LIN {X 0,Y 423.097,Z 216.346,A -85,B 0,C 180,E1 -10151.866,E2 -10151.866} C_VEL
LIN {X 0,Y 422.298,Z 296.98,A -85,B 0,C 180,E1 -10153.256,E2 -10153.256} C_VEL
LIN {X 0,Y 421.712,Z 310.923,A -85,B 0,C 180,E1 -10153.699,E2 -10153.699} C_VEL
LIN {X 0,Y 421.172,Z 322.869,A -85,B 0,C 180,E1 -10154.268,E2 -10154.268} C_VEL
LIN {X 0,Y 420.503,Z 334.151,A -85,B 0,C 180,E1 -10154.987,E2 -10154.987} C_VEL
LIN {X 0,Y 419.836,Z 344.931,A -85,B 0,C 180,E1 -10155.867,E2 -10155.867} C_VEL
LIN {X 0,Y 419.115,Z 356.382,A -85,B 0,C 180,E1 -10157.042,E2 -10157.042} C_VEL
LIN {X 0,Y 418.563,Z 364.963,A -85,B 0,C 180,E1 -10158.131,E2 -10158.131} C_VEL
LIN {X 0,Y 417.991,Z 372.886,A -85,B 0,C 180,E1 -10159.343,E2 -10159.343} C_VEL
LIN {X 0,Y 417.563,Z 380.623,A -85,B 0,C 180,E1 -10160.8,E2 -10160.8} C_VEL
LIN {X 0,Y 417.305,Z 386.839,A -85,B 0,C 180,E1 -10162.258,E2 -10162.258} C_VEL
LIN {X 0,Y 417.13,Z 391.886,A -85,B 0,C 180,E1 -10163.753,E2 -10163.753} C_VEL
LIN {X 0,Y 417.134,Z 395.569,A -85,B 0,C 180,E1 -10165.169,E2 -10165.169} C_VEL
LIN {X 0,Y 417.042,Z 397.521,A -85,B 0,C 180,E1 -10166.136,E2 -10166.136} C_VEL
LIN {X 0,Y 417.114,Z 399.058,A -85,B 0,C 180,E1 -10167.104,E2 -10167.104} C_VEL
LIN {X 0,Y 417.095,Z 400.134,A -85,B 0,C 180,E1 -10168.07,E2 -10168.07} C_VEL
LIN {X 0,Y 417.059,Z 401.099,A -85,B 0,C 180,E1 -10170.001,E2 -10170.001} C_VEL
LIN {X 0,Y 417.06,Z 400.999,A -85,B 0,C 180,E1 -10170.966,E2 -10170.966} C_VEL
LIN {X 0,Y 417.092,Z 400.466,A -85,B 0,C 180,E1 -10171.932,E2 -10171.932} C_VEL
LIN {X 0,Y 417.074,Z 399.531,A -85,B 0,C 180,E1 -10172.899,E2 -10172.899} C_VEL
LIN {X 0,Y 417.101,Z 396.464,A -85,B 0,C 180,E1 -10174.834,E2 -10174.834} C_VEL
LIN {X 0,Y 417.064,Z 393.308,A -85,B 0,C 180,E1 -10176.163,E2 -10176.163} C_VEL
LIN {X 0,Y 417.325,Z 388.427,A -85,B 0,C 180,E1 -10177.743,E2 -10177.743} C_VEL
LIN {X 0,Y 417.698,Z 381.536,A -85,B 0,C 180,E1 -10179.443,E2 -10179.443} C_VEL
LIN {X 0,Y 418.217,Z 374.083,A -85,B 0,C 180,E1 -10180.898,E2 -10180.898} C_VEL
LIN {X 0,Y 418.892,Z 366.504,A -85,B 0,C 180,E1 -10182.107,E2 -10182.107} C_VEL
LIN {X 0,Y 419.495,Z 357.34,A -85,B 0,C 180,E1 -10183.319,E2 -10183.319} C_VEL
LIN {X 0,Y 420.276,Z 347.151,A -85,B 0,C 180,E1 -10184.407,E2 -10184.407} C_VEL
LIN {X 0,Y 421.16,Z 335.937,A -85,B 0,C 180,E1 -10185.362,E2 -10185.362} C_VEL
LIN {X 0,Y 422.016,Z 323.303,A -85,B 0,C 180,E1 -10186.198,E2 -10186.198} C_VEL
LIN {X 0,Y 422.766,Z 310.212,A -85,B 0,C 180,E1 -10186.82,E2 -10186.82} C_VEL
LIN {X 0,Y 423.348,Z 297.267,A -85,B 0,C 180,E1 -10187.232,E2 -10187.232} C_VEL
LIN {X 0,Y 424.197,Z 227.472,A -85,B 0,C 180,E1 -10188.452,E2 -10188.452} C_VEL
LIN {X 0,Y 424.203,Z 214.443,A -85,B 0,C 180,E1 -10188.682,E2 -10188.682} C_VEL
LIN {X 0,Y 420.161,Z 189.661,A -85,B 0,C 180,E1 -10189.327,E2 -10189.327} C_VEL
LIN {X 0,Y 419.865,Z 187.56,A -85,B 0,C 180,E1 -10189.403,E2 -10189.403} C_VEL
LIN {X 0,Y 421.208,Z 166.448,A -85,B 0,C 180,E1 -10193.408,E2 -10193.408} C_VEL
LIN {X 0,Y 421.73,Z 158.765,A -85,B 0,C 180,E1 -10194.885,E2 -10194.885} C_VEL
LIN {X 0,Y 420.332,Z 150.718,A -85,B 0,C 180,E1 -10196.569,E2 -10196.569} C_VEL
LIN {X 0,Y 418.298,Z 141.385,A -85,B 0,C 180,E1 -10198.61,E2 -10198.61} C_VEL
LIN {X 0,Y 418.214,Z 141.395,A -85,B 0,C 180,E1 -10201.396,E2 -10201.396} C_VEL
LIN {X 0,Y 418.268,Z 141.381,A -85,B 0,C 180,E1 -10204.58,E2 -10204.58} C_VEL
LIN {X 0,Y 418.226,Z 141.39,A -85,B 0,C 180,E1 -10207.833,E2 -10207.833} C_VEL
LIN {X 0,Y 418.221,Z 141.387,A -85,B 0,C 180,E1 -10210.949,E2 -10210.949} C_VEL
LIN {X 0,Y 418.211,Z 141.392,A -85,B 0,C 180,E1 -10213.729,E2 -10213.729} C_VEL
LIN {X 0,Y 418.208,Z 141.389,A -85,B 0,C 180,E1 -10216.448,E2 -10216.448} C_VEL
LIN {X 0,Y 418.211,Z 141.393,A -85,B 0,C 180,E1 -10219.133,E2 -10219.133} C_VEL
LIN {X 0,Y 418.24,Z 141.388,A -85,B 0,C 180,E1 -10222.776,E2 -10222.776} C_VEL
LIN {X 0,Y 418.234,Z 141.387,A -85,B 0,C 180,E1 -10226.321,E2 -10226.321} C_VEL
LIN {X 0,Y 418.242,Z 141.384,A -85,B 0,C 180,E1 -10229.728,E2 -10229.728} C_VEL
LIN {X 0,Y 418.222,Z 141.391,A -85,B 0,C 180,E1 -10233.017,E2 -10233.017} C_VEL
LIN {X 0,Y 418.258,Z 141.384,A -85,B 0,C 180,E1 -10236.217,E2 -10236.217} C_VEL
LIN {X 0,Y 418.247,Z 141.38,A -85,B 0,C 180,E1 -10239.337,E2 -10239.337} C_VEL
LIN {X 0,Y 418.256,Z 141.385,A -85,B 0,C 180,E1 -10242.395,E2 -10242.395} C_VEL
LIN {X 0,Y 418.263,Z 141.375,A -85,B 0,C 180,E1 -10245.402,E2 -10245.402} C_VEL
LIN {X 0,Y 418.352,Z 141.368,A -85,B 0,C 180,E1 -10247.386,E2 -10247.386} C_VEL
LIN {X 0,Y 418.366,Z 141.361,A -85,B 0,C 180,E1 -10251.304,E2 -10251.304} C_VEL
LIN {X 0,Y 418.467,Z 141.361,A -85,B 0,C 180,E1 -10254.217,E2 -10254.217} C_VEL
LIN {X 0,Y 418.532,Z 141.347,A -85,B 0,C 180,E1 -10258.076,E2 -10258.076} C_VEL
LIN {X 0,Y 418.405,Z 141.363,A -85,B 0,C 180,E1 -10260.963,E2 -10260.963} C_VEL
LIN {X 0,Y 418.468,Z 141.348,A -85,B 0,C 180,E1 -10262.888,E2 -10262.888} C_VEL
LIN {X 0,Y 418.44,Z 141.359,A -85,B 0,C 180,E1 -10266.478,E2 -10266.478} C_VEL
LIN {X 0,Y 418.377,Z 141.359,A -85,B 0,C 180,E1 -10268.696,E2 -10268.696} C_VEL
LIN {X 0,Y 418.314,Z 141.38,A -85,B 0,C 180,E1 -10271.631,E2 -10271.631} C_VEL
LIN {X 0,Y 418.299,Z 141.37,A -85,B 0,C 180,E1 -10274.597,E2 -10274.597} C_VEL
LIN {X 0,Y 418.28,Z 141.381,A -85,B 0,C 180,E1 -10277.604,E2 -10277.604} C_VEL
LIN {X 0,Y 418.251,Z 141.381,A -85,B 0,C 180,E1 -10280.663,E2 -10280.663} C_VEL
LIN {X 0,Y 418.274,Z 141.376,A -85,B 0,C 180,E1 -10283.782,E2 -10283.782} C_VEL
LIN {X 0,Y 418.268,Z 141.385,A -85,B 0,C 180,E1 -10287.059,E2 -10287.059} C_VEL
LIN {X 0,Y 418.244,Z 141.384,A -85,B 0,C 180,E1 -10290.272,E2 -10290.272} C_VEL
LIN {X 0,Y 418.249,Z 141.382,A -85,B 0,C 180,E1 -10293.677,E2 -10293.677} C_VEL
LIN {X 0,Y 418.241,Z 141.385,A -85,B 0,C 180,E1 -10297.224,E2 -10297.224} C_VEL
LIN {X 0,Y 418.245,Z 141.38,A -85,B 0,C 180,E1 -10299.683,E2 -10299.683} C_VEL
LIN {X 0,Y 418.232,Z 141.38,A -85,B 0,C 180,E1 -10302.321,E2 -10302.321} C_VEL
LIN {X 0,Y 418.239,Z 141.384,A -85,B 0,C 180,E1 -10305.109,E2 -10305.109} C_VEL
LIN {X 0,Y 418.237,Z 141.386,A -85,B 0,C 180,E1 -10307.766,E2 -10307.766} C_VEL
LIN {X 0,Y 418.246,Z 141.386,A -85,B 0,C 180,E1 -10310.621,E2 -10310.621} C_VEL
LIN {X 0,Y 418.247,Z 141.389,A -85,B 0,C 180,E1 -10313.976,E2 -10313.976} C_VEL
LIN {X 0,Y 418.262,Z 141.383,A -85,B 0,C 180,E1 -10317.156,E2 -10317.156} C_VEL
LIN {X 0,Y 418.273,Z 141.384,A -85,B 0,C 180,E1 -10320.895,E2 -10320.895} C_VEL
LIN {X 0,Y 418.345,Z 141.524,A -85,B 0,C 180,E1 -10323.025,E2 -10323.025} C_VEL
LIN {X 0,Y 420.17,Z 150.792,A -85,B 0,C 180,E1 -10325.281,E2 -10325.281} C_VEL
LIN {X 0,Y 420.345,Z 152.604,A -85,B 0,C 180,E1 -10325.696,E2 -10325.696} C_VEL
LIN {X 0,Y 424.762,Z 171.221,A -85,B 0,C 180,E1 -10326.26,E2 -10326.26} C_VEL
LIN {X 0,Y 423.727,Z 259.847,A -85,B 0,C 180,E1 -10327.799,E2 -10327.799} C_VEL
LIN {X 0,Y 423.245,Z 273.544,A -85,B 0,C 180,E1 -10328.237,E2 -10328.237} C_VEL
LIN {X 0,Y 422.763,Z 285.058,A -85,B 0,C 180,E1 -10328.786,E2 -10328.786} C_VEL
LIN {X 0,Y 422.155,Z 296.809,A -85,B 0,C 180,E1 -10329.536,E2 -10329.536} C_VEL
LIN {X 0,Y 421.289,Z 308.537,A -85,B 0,C 180,E1 -10330.509,E2 -10330.509} C_VEL
LIN {X 0,Y 420.515,Z 319.047,A -85,B 0,C 180,E1 -10331.611,E2 -10331.611} C_VEL
LIN {X 0,Y 419.859,Z 328.587,A -85,B 0,C 180,E1 -10332.858,E2 -10332.858} C_VEL
LIN {X 0,Y 419.159,Z 336.843,A -85,B 0,C 180,E1 -10334.188,E2 -10334.188} C_VEL
LIN {X 0,Y 418.482,Z 344.233,A -85,B 0,C 180,E1 -10335.657,E2 -10335.657} C_VEL
LIN {X 0,Y 417.937,Z 350.995,A -85,B 0,C 180,E1 -10337.372,E2 -10337.372} C_VEL
LIN {X 0,Y 417.623,Z 355.433,A -85,B 0,C 180,E1 -10338.84,E2 -10338.84} C_VEL
LIN {X 0,Y 417.337,Z 358.788,A -85,B 0,C 180,E1 -10340.304,E2 -10340.304} C_VEL
LIN {X 0,Y 417.213,Z 361.303,A -85,B 0,C 180,E1 -10341.946,E2 -10341.946} C_VEL
LIN {X 0,Y 416.513,Z 362.24,A -85,B 0,C 180,E1 -10342.743,E2 -10342.743} C_VEL
LIN {X 0,Y 413.581,Z 363.208,A -85,B 0,C 180,E1 -10344.045,E2 -10344.045} C_VEL
LIN {X 0,Y 411.127,Z 363.394,A -85,B 0,C 180,E1 -10345.101,E2 -10345.101} C_VEL
LIN {X 0,Y 410.094,Z 363.129,A -85,B 0,C 180,E1 -10345.917,E2 -10345.917} C_VEL
LIN {X 0,Y 410.022,Z 362.954,A -85,B 0,C 180,E1 -10346.193,E2 -10346.193} C_VEL
LIN {X 0,Y 410.105,Z 362.339,A -85,B 0,C 180,E1 -10347.052,E2 -10347.052} C_VEL
LIN {X 0,Y 410.075,Z 361.229,A -85,B 0,C 180,E1 -10348.035,E2 -10348.035} C_VEL
LIN {X 0,Y 410.201,Z 357.742,A -85,B 0,C 180,E1 -10349.999,E2 -10349.999} C_VEL
LIN {X 0,Y 410.379,Z 353.97,A -85,B 0,C 180,E1 -10351.471,E2 -10351.471} C_VEL
LIN {X 0,Y 410.654,Z 349.089,A -85,B 0,C 180,E1 -10352.942,E2 -10352.942} C_VEL
LIN {X 0,Y 411.139,Z 342.947,A -85,B 0,C 180,E1 -10354.411,E2 -10354.411} C_VEL
LIN {X 0,Y 411.719,Z 335.291,A -85,B 0,C 180,E1 -10355.878,E2 -10355.878} C_VEL
LIN {X 0,Y 412.361,Z 327.463,A -85,B 0,C 180,E1 -10357.097,E2 -10357.097} C_VEL
LIN {X 0,Y 413.07,Z 317.923,A -85,B 0,C 180,E1 -10358.314,E2 -10358.314} C_VEL
LIN {X 0,Y 413.815,Z 307.327,A -85,B 0,C 180,E1 -10359.407,E2 -10359.407} C_VEL
LIN {X 0,Y 414.433,Z 296.178,A -85,B 0,C 180,E1 -10360.323,E2 -10360.323} C_VEL
LIN {X 0,Y 414.947,Z 283.723,A -85,B 0,C 180,E1 -10361.107,E2 -10361.107} C_VEL
LIN {X 0,Y 415.398,Z 271.188,A -85,B 0,C 180,E1 -10361.682,E2 -10361.682} C_VEL
LIN {X 0,Y 415.689,Z 257.936,A -85,B 0,C 180,E1 -10362.076,E2 -10362.076} C_VEL
LIN {X 0,Y 416.741,Z 172.858,A -85,B 0,C 180,E1 -10363.547,E2 -10363.547} C_VEL
LIN {X 0,Y 412.858,Z 152.57,A -85,B 0,C 180,E1 -10364.097,E2 -10364.097} C_VEL
LIN {X 0,Y 412.536,Z 148.394,A -85,B 0,C 180,E1 -10365.057,E2 -10365.057} C_VEL
LIN {X 0,Y 411.291,Z 142.256,A -85,B 0,C 180,E1 -10366.551,E2 -10366.551} C_VEL
LIN {X 0,Y 411.231,Z 142.263,A -85,B 0,C 180,E1 -10369.985,E2 -10369.985} C_VEL
LIN {X 0,Y 411.195,Z 142.262,A -85,B 0,C 180,E1 -10373.147,E2 -10373.147} C_VEL
LIN {X 0,Y 411.236,Z 142.261,A -85,B 0,C 180,E1 -10376.38,E2 -10376.38} C_VEL
LIN {X 0,Y 411.198,Z 142.263,A -85,B 0,C 180,E1 -10379.711,E2 -10379.711} C_VEL
LIN {X 0,Y 411.204,Z 142.261,A -85,B 0,C 180,E1 -10383.154,E2 -10383.154} C_VEL
LIN {X 0,Y 411.189,Z 142.265,A -85,B 0,C 180,E1 -10386.551,E2 -10386.551} C_VEL
LIN {X 0,Y 411.213,Z 142.264,A -85,B 0,C 180,E1 -10389.727,E2 -10389.727} C_VEL
LIN {X 0,Y 411.168,Z 142.266,A -85,B 0,C 180,E1 -10393.132,E2 -10393.132} C_VEL
LIN {X 0,Y 411.161,Z 142.271,A -85,B 0,C 180,E1 -10395.88,E2 -10395.88} C_VEL
LIN {X 0,Y 411.156,Z 142.267,A -85,B 0,C 180,E1 -10398.771,E2 -10398.771} C_VEL
LIN {X 0,Y 411.184,Z 142.266,A -85,B 0,C 180,E1 -10402.025,E2 -10402.025} C_VEL
LIN {X 0,Y 411.196,Z 142.266,A -85,B 0,C 180,E1 -10405.665,E2 -10405.665} C_VEL
LIN {X 0,Y 411.18,Z 142.267,A -85,B 0,C 180,E1 -10409.151,E2 -10409.151} C_VEL
LIN {X 0,Y 411.249,Z 142.256,A -85,B 0,C 180,E1 -10412.521,E2 -10412.521} C_VEL
LIN {X 0,Y 411.201,Z 142.265,A -85,B 0,C 180,E1 -10415.783,E2 -10415.783} C_VEL
LIN {X 0,Y 411.185,Z 142.266,A -85,B 0,C 180,E1 -10418.965,E2 -10418.965} C_VEL
LIN {X 0,Y 411.232,Z 142.259,A -85,B 0,C 180,E1 -10422.084,E2 -10422.084} C_VEL
LIN {X 0,Y 411.24,Z 142.261,A -85,B 0,C 180,E1 -10425.146,E2 -10425.146} C_VEL
LIN {X 0,Y 411.27,Z 142.254,A -85,B 0,C 180,E1 -10428.167,E2 -10428.167} C_VEL
LIN {X 0,Y 411.306,Z 142.252,A -85,B 0,C 180,E1 -10431.154,E2 -10431.154} C_VEL
LIN {X 0,Y 411.405,Z 142.237,A -85,B 0,C 180,E1 -10434.117,E2 -10434.117} C_VEL
LIN {X 0,Y 411.489,Z 142.226,A -85,B 0,C 180,E1 -10438.042,E2 -10438.042} C_VEL
LIN {X 0,Y 411.364,Z 142.245,A -85,B 0,C 180,E1 -10440.979,E2 -10440.979} C_VEL
LIN {X 0,Y 411.416,Z 142.238,A -85,B 0,C 180,E1 -10442.937,E2 -10442.937} C_VEL
LIN {X 0,Y 411.418,Z 142.235,A -85,B 0,C 180,E1 -10445.883,E2 -10445.883} C_VEL
LIN {X 0,Y 411.306,Z 142.252,A -85,B 0,C 180,E1 -10448.846,E2 -10448.846} C_VEL
LIN {X 0,Y 411.27,Z 142.254,A -85,B 0,C 180,E1 -10451.833,E2 -10451.833} C_VEL
LIN {X 0,Y 411.245,Z 142.26,A -85,B 0,C 180,E1 -10454.853,E2 -10454.853} C_VEL
LIN {X 0,Y 411.233,Z 142.258,A -85,B 0,C 180,E1 -10457.916,E2 -10457.916} C_VEL
LIN {X 0,Y 411.185,Z 142.267,A -85,B 0,C 180,E1 -10461.035,E2 -10461.035} C_VEL
LIN {X 0,Y 411.2,Z 142.264,A -85,B 0,C 180,E1 -10464.217,E2 -10464.217} C_VEL
LIN {X 0,Y 411.248,Z 142.256,A -85,B 0,C 180,E1 -10467.478,E2 -10467.478} C_VEL
LIN {X 0,Y 411.18,Z 142.267,A -85,B 0,C 180,E1 -10470.848,E2 -10470.848} C_VEL
LIN {X 0,Y 411.195,Z 142.266,A -85,B 0,C 180,E1 -10474.335,E2 -10474.335} C_VEL
LIN {X 0,Y 411.183,Z 142.266,A -85,B 0,C 180,E1 -10477.975,E2 -10477.975} C_VEL
LIN {X 0,Y 411.155,Z 142.267,A -85,B 0,C 180,E1 -10481.229,E2 -10481.229} C_VEL
LIN {X 0,Y 411.168,Z 142.269,A -85,B 0,C 180,E1 -10484.492,E2 -10484.492} C_VEL
LIN {X 0,Y 411.171,Z 142.271,A -85,B 0,C 180,E1 -10488.196,E2 -10488.196} C_VEL
LIN {X 0,Y 411.217,Z 142.26,A -85,B 0,C 180,E1 -10490.778,E2 -10490.778} C_VEL
LIN {X 0,Y 411.193,Z 142.264,A -85,B 0,C 180,E1 -10494.472,E2 -10494.472} C_VEL
LIN {X 0,Y 411.203,Z 142.26,A -85,B 0,C 180,E1 -10496.875,E2 -10496.875} C_VEL
LIN {X 0,Y 411.23,Z 142.263,A -85,B 0,C 180,E1 -10500.645,E2 -10500.645} C_VEL
LIN {X 0,Y 411.295,Z 142.381,A -85,B 0,C 180,E1 -10502.05,E2 -10502.05} C_VEL
LIN {X 0,Y 413.922,Z 155.94,A -85,B 0,C 180,E1 -10504.884,E2 -10504.884} C_VEL
LIN {X 0,Y 414.049,Z 160.059,A -85,B 0,C 180,E1 -10505.695,E2 -10505.695} C_VEL
LIN {X 0,Y 412.864,Z 177.718,A -85,B 0,C 180,E1 -10509.056,E2 -10509.056} C_VEL
LIN {X 0,Y 412.362,Z 187.731,A -85,B 0,C 180,E1 -10510.925,E2 -10510.925} C_VEL
LIN {X 0,Y 416.291,Z 216.452,A -85,B 0,C 180,E1 -10511.597,E2 -10511.597} C_VEL
LIN {X 0,Y 415.449,Z 296.703,A -85,B 0,C 180,E1 -10513.003,E2 -10513.003} C_VEL
LIN {X 0,Y 414.83,Z 310.629,A -85,B 0,C 180,E1 -10513.452,E2 -10513.452} C_VEL
LIN {X 0,Y 414.247,Z 323.112,A -85,B 0,C 180,E1 -10514.061,E2 -10514.061} C_VEL
LIN {X 0,Y 413.503,Z 335.041,A -85,B 0,C 180,E1 -10514.853,E2 -10514.853} C_VEL
LIN {X 0,Y 412.729,Z 346.51,A -85,B 0,C 180,E1 -10515.832,E2 -10515.832} C_VEL
LIN {X 0,Y 412.066,Z 357.099,A -85,B 0,C 180,E1 -10516.97,E2 -10516.97} C_VEL
LIN {X 0,Y 411.452,Z 366.135,A -85,B 0,C 180,E1 -10518.173,E2 -10518.173} C_VEL
LIN {X 0,Y 410.775,Z 375.155,A -85,B 0,C 180,E1 -10519.652,E2 -10519.652} C_VEL
LIN {X 0,Y 410.4,Z 382.423,A -85,B 0,C 180,E1 -10521.135,E2 -10521.135} C_VEL
LIN {X 0,Y 410.171,Z 388.22,A -85,B 0,C 180,E1 -10522.618,E2 -10522.618} C_VEL
LIN {X 0,Y 410.002,Z 392.777,A -85,B 0,C 180,E1 -10524.098,E2 -10524.098} C_VEL
LIN {X 0,Y 410.041,Z 395.183,A -85,B 0,C 180,E1 -10525.085,E2 -10525.085} C_VEL
LIN {X 0,Y 409.959,Z 397.146,A -85,B 0,C 180,E1 -10526.069,E2 -10526.069} C_VEL
LIN {X 0,Y 410.011,Z 398.696,A -85,B 0,C 180,E1 -10527.053,E2 -10527.053} C_VEL
LIN {X 0,Y 410.023,Z 399.789,A -85,B 0,C 180,E1 -10528.036,E2 -10528.036} C_VEL
LIN {X 0,Y 409.978,Z 400.772,A -85,B 0,C 180,E1 -10530.001,E2 -10530.001} C_VEL
LIN {X 0,Y 409.982,Z 400.682,A -85,B 0,C 180,E1 -10530.983,E2 -10530.983} C_VEL
LIN {X 0,Y 410.019,Z 400.166,A -85,B 0,C 180,E1 -10531.965,E2 -10531.965} C_VEL
LIN {X 0,Y 409.971,Z 399.239,A -85,B 0,C 180,E1 -10532.949,E2 -10532.949} C_VEL
LIN {X 0,Y 410.008,Z 396.194,A -85,B 0,C 180,E1 -10534.917,E2 -10534.917} C_VEL
LIN {X 0,Y 409.999,Z 392.73,A -85,B 0,C 180,E1 -10536.397,E2 -10536.397} C_VEL
LIN {X 0,Y 410.266,Z 388.196,A -85,B 0,C 180,E1 -10537.878,E2 -10537.878} C_VEL
LIN {X 0,Y 410.654,Z 381.341,A -85,B 0,C 180,E1 -10539.606,E2 -10539.606} C_VEL
LIN {X 0,Y 411.219,Z 373.917,A -85,B 0,C 180,E1 -10541.086,E2 -10541.086} C_VEL
LIN {X 0,Y 412.045,Z 364.711,A -85,B 0,C 180,E1 -10542.561,E2 -10542.561} C_VEL
LIN {X 0,Y 412.7,Z 355.159,A -85,B 0,C 180,E1 -10543.793,E2 -10543.793} C_VEL
LIN {X 0,Y 413.608,Z 344.588,A -85,B 0,C 180,E1 -10544.893,E2 -10544.893} C_VEL
LIN {X 0,Y 414.57,Z 332.794,A -85,B 0,C 180,E1 -10545.865,E2 -10545.865} C_VEL
LIN {X 0,Y 415.393,Z 320.17,A -85,B 0,C 180,E1 -10546.653,E2 -10546.653} C_VEL
LIN {X 0,Y 416.117,Z 307.584,A -85,B 0,C 180,E1 -10547.224,E2 -10547.224} C_VEL
LIN {X 0,Y 416.707,Z 294.35,A -85,B 0,C 180,E1 -10547.61,E2 -10547.61} C_VEL
LIN {X 0,Y 417.568,Z 215.601,A -85,B 0,C 180,E1 -10548.994,E2 -10548.994} C_VEL
LIN {X 0,Y 413.767,Z 191.967,A -85,B 0,C 180,E1 -10549.621,E2 -10549.621} C_VEL
LIN {X 0,Y 412.962,Z 187.289,A -85,B 0,C 180,E1 -10549.761,E2 -10549.761} C_VEL
LIN {X 0,Y 414.195,Z 168.849,A -85,B 0,C 180,E1 -10553.32,E2 -10553.32} C_VEL
LIN {X 0,Y 414.816,Z 159.947,A -85,B 0,C 180,E1 -10555.06,E2 -10555.06} C_VEL
LIN {X 0,Y 413.088,Z 150.562,A -85,B 0,C 180,E1 -10557.072,E2 -10557.072} C_VEL
LIN {X 0,Y 411.23,Z 142.266,A -85,B 0,C 180,E1 -10558.951,E2 -10558.951} C_VEL
LIN {X 0,Y 411.169,Z 142.275,A -85,B 0,C 180,E1 -10561.998,E2 -10561.998} C_VEL
LIN {X 0,Y 411.213,Z 142.259,A -85,B 0,C 180,E1 -10564.879,E2 -10564.879} C_VEL
LIN {X 0,Y 411.201,Z 142.262,A -85,B 0,C 180,E1 -10568.168,E2 -10568.168} C_VEL
LIN {X 0,Y 411.163,Z 142.268,A -85,B 0,C 180,E1 -10571.228,E2 -10571.228} C_VEL
LIN {X 0,Y 411.178,Z 142.264,A -85,B 0,C 180,E1 -10574.491,E2 -10574.491} C_VEL
LIN {X 0,Y 411.17,Z 142.266,A -85,B 0,C 180,E1 -10578.194,E2 -10578.194} C_VEL
LIN {X 0,Y 411.196,Z 142.264,A -85,B 0,C 180,E1 -10581.833,E2 -10581.833} C_VEL
LIN {X 0,Y 411.204,Z 142.266,A -85,B 0,C 180,E1 -10585.123,E2 -10585.123} C_VEL
LIN {X 0,Y 411.166,Z 142.266,A -85,B 0,C 180,E1 -10588.003,E2 -10588.003} C_VEL
LIN {X 0,Y 411.179,Z 142.265,A -85,B 0,C 180,E1 -10591.407,E2 -10591.407} C_VEL
LIN {X 0,Y 411.213,Z 142.264,A -85,B 0,C 180,E1 -10594.934,E2 -10594.934} C_VEL
LIN {X 0,Y 411.202,Z 142.261,A -85,B 0,C 180,E1 -10597.913,E2 -10597.913} C_VEL
LIN {X 0,Y 411.215,Z 142.258,A -85,B 0,C 180,E1 -10601.051,E2 -10601.051} C_VEL
LIN {X 0,Y 411.21,Z 142.263,A -85,B 0,C 180,E1 -10604.13,E2 -10604.13} C_VEL
LIN {X 0,Y 411.302,Z 142.247,A -85,B 0,C 180,E1 -10607.166,E2 -10607.166} C_VEL
LIN {X 0,Y 411.272,Z 142.253,A -85,B 0,C 180,E1 -10610.161,E2 -10610.161} C_VEL
LIN {X 0,Y 411.389,Z 142.236,A -85,B 0,C 180,E1 -10613.132,E2 -10613.132} C_VEL
LIN {X 0,Y 411.281,Z 142.251,A -85,B 0,C 180,E1 -10615.099,E2 -10615.099} C_VEL
LIN {X 0,Y 411.5,Z 142.222,A -85,B 0,C 180,E1 -10618.043,E2 -10618.043} C_VEL
LIN {X 0,Y 411.376,Z 142.239,A -85,B 0,C 180,E1 -10620.979,E2 -10620.979} C_VEL
LIN {X 0,Y 411.427,Z 142.225,A -85,B 0,C 180,E1 -10622.938,E2 -10622.938} C_VEL
LIN {X 0,Y 411.39,Z 142.237,A -85,B 0,C 180,E1 -10626.475,E2 -10626.475} C_VEL
LIN {X 0,Y 411.318,Z 142.238,A -85,B 0,C 180,E1 -10628.846,E2 -10628.846} C_VEL
LIN {X 0,Y 411.283,Z 142.253,A -85,B 0,C 180,E1 -10631.833,E2 -10631.833} C_VEL
LIN {X 0,Y 411.257,Z 142.248,A -85,B 0,C 180,E1 -10634.853,E2 -10634.853} C_VEL
LIN {X 0,Y 411.246,Z 142.254,A -85,B 0,C 180,E1 -10637.916,E2 -10637.916} C_VEL
LIN {X 0,Y 411.197,Z 142.263,A -85,B 0,C 180,E1 -10641.034,E2 -10641.034} C_VEL
LIN {X 0,Y 411.205,Z 142.256,A -85,B 0,C 180,E1 -10644.217,E2 -10644.217} C_VEL
LIN {X 0,Y 411.21,Z 142.26,A -85,B 0,C 180,E1 -10647.481,E2 -10647.481} C_VEL
LIN {X 0,Y 411.191,Z 142.269,A -85,B 0,C 180,E1 -10650.848,E2 -10650.848} C_VEL
LIN {X 0,Y 411.207,Z 142.262,A -85,B 0,C 180,E1 -10654.334,E2 -10654.334} C_VEL
LIN {X 0,Y 411.192,Z 142.263,A -85,B 0,C 180,E1 -10657.974,E2 -10657.974} C_VEL
LIN {X 0,Y 411.166,Z 142.254,A -85,B 0,C 180,E1 -10661.228,E2 -10661.228} C_VEL
LIN {X 0,Y 411.179,Z 142.267,A -85,B 0,C 180,E1 -10664.49,E2 -10664.49} C_VEL
LIN {X 0,Y 411.176,Z 142.269,A -85,B 0,C 180,E1 -10668.194,E2 -10668.194} C_VEL
LIN {X 0,Y 411.211,Z 142.261,A -85,B 0,C 180,E1 -10670.775,E2 -10670.775} C_VEL
LIN {X 0,Y 411.202,Z 142.265,A -85,B 0,C 180,E1 -10674.471,E2 -10674.471} C_VEL
LIN {X 0,Y 411.211,Z 142.261,A -85,B 0,C 180,E1 -10676.873,E2 -10676.873} C_VEL
LIN {X 0,Y 411.237,Z 142.26,A -85,B 0,C 180,E1 -10680.644,E2 -10680.644} C_VEL
LIN {X 0,Y 411.271,Z 142.275,A -85,B 0,C 180,E1 -10682.699,E2 -10682.699} C_VEL
LIN {X 0,Y 413.324,Z 152.796,A -85,B 0,C 180,E1 -10685.296,E2 -10685.296} C_VEL
LIN {X 0,Y 416.305,Z 163.879,A -85,B 0,C 180,E1 -10685.682,E2 -10685.682} C_VEL
LIN {X 0,Y 418.173,Z 172.485,A -85,B 0,C 180,E1 -10685.938,E2 -10685.938} C_VEL
LIN {X 0,Y 417.039,Z 260.378,A -85,B 0,C 180,E1 -10687.488,E2 -10687.488} C_VEL
LIN {X 0,Y 416.545,Z 273.617,A -85,B 0,C 180,E1 -10687.917,E2 -10687.917} C_VEL
LIN {X 0,Y 416.027,Z 285.707,A -85,B 0,C 180,E1 -10688.503,E2 -10688.503} C_VEL
LIN {X 0,Y 415.443,Z 296.354,A -85,B 0,C 180,E1 -10689.19,E2 -10689.19} C_VEL
LIN {X 0,Y 414.552,Z 308.269,A -85,B 0,C 180,E1 -10690.179,E2 -10690.179} C_VEL
LIN {X 0,Y 413.726,Z 318.88,A -85,B 0,C 180,E1 -10691.298,E2 -10691.298} C_VEL
LIN {X 0,Y 413.035,Z 328.056,A -85,B 0,C 180,E1 -10692.496,E2 -10692.496} C_VEL
LIN {X 0,Y 412.233,Z 336.857,A -85,B 0,C 180,E1 -10693.916,E2 -10693.916} C_VEL
LIN {X 0,Y 411.524,Z 344.301,A -85,B 0,C 180,E1 -10695.409,E2 -10695.409} C_VEL
LIN {X 0,Y 410.925,Z 351.134,A -85,B 0,C 180,E1 -10697.153,E2 -10697.153} C_VEL
LIN {X 0,Y 410.584,Z 355.615,A -85,B 0,C 180,E1 -10698.647,E2 -10698.647} C_VEL
LIN {X 0,Y 410.269,Z 359.01,A -85,B 0,C 180,E1 -10700.136,E2 -10700.136} C_VEL
LIN {X 0,Y 410.131,Z 361.72,A -85,B 0,C 180,E1 -10701.933,E2 -10701.933} C_VEL
LIN {X 0,Y 410.128,Z 363.135,A -85,B 0,C 180,E1 -10703.668,E2 -10703.668} C_VEL
LIN {X 0,Y 410.061,Z 363.364,A -85,B 0,C 180,E1 -10705.083,E2 -10705.083} C_VEL
LIN {X 0,Y 410.022,Z 362.954,A -85,B 0,C 180,E1 -10706.193,E2 -10706.193} C_VEL
LIN {X 0,Y 409.378,Z 362.408,A -85,B 0,C 180,E1 -10707.008,E2 -10707.008} C_VEL
LIN {X 0,Y 406.531,Z 360.981,A -85,B 0,C 180,E1 -10708.328,E2 -10708.328} C_VEL
LIN {X 0,Y 404.161,Z 359.374,A -85,B 0,C 180,E1 -10709.381,E2 -10709.381} C_VEL
LIN {X 0,Y 403.217,Z 357.79,A -85,B 0,C 180,E1 -10710.184,E2 -10710.184} C_VEL
LIN {X 0,Y 403.181,Z 357.166,A -85,B 0,C 180,E1 -10710.453,E2 -10710.453} C_VEL
LIN {X 0,Y 403.379,Z 352.98,A -85,B 0,C 180,E1 -10711.996,E2 -10711.996} C_VEL
LIN {X 0,Y 403.864,Z 346.734,A -85,B 0,C 180,E1 -10713.741,E2 -10713.741} C_VEL
LIN {X 0,Y 404.389,Z 339.941,A -85,B 0,C 180,E1 -10715.234,E2 -10715.234} C_VEL
LIN {X 0,Y 404.982,Z 333.002,A -85,B 0,C 180,E1 -10716.476,E2 -10716.476} C_VEL
LIN {X 0,Y 405.626,Z 324.654,A -85,B 0,C 180,E1 -10717.716,E2 -10717.716} C_VEL
LIN {X 0,Y 406.431,Z 314.339,A -85,B 0,C 180,E1 -10718.952,E2 -10718.952} C_VEL
LIN {X 0,Y 407.161,Z 302.627,A -85,B 0,C 180,E1 -10720.074,E2 -10720.074} C_VEL
LIN {X 0,Y 407.799,Z 291.16,A -85,B 0,C 180,E1 -10720.927,E2 -10720.927} C_VEL
LIN {X 0,Y 408.284,Z 279.152,A -85,B 0,C 180,E1 -10721.605,E2 -10721.605} C_VEL
LIN {X 0,Y 408.737,Z 266.047,A -85,B 0,C 180,E1 -10722.127,E2 -10722.127} C_VEL
LIN {X 0,Y 408.942,Z 253.349,A -85,B 0,C 180,E1 -10722.436,E2 -10722.436} C_VEL
LIN {X 0,Y 409.873,Z 172.692,A -85,B 0,C 180,E1 -10723.845,E2 -10723.845} C_VEL
LIN {X 0,Y 405.923,Z 152.861,A -85,B 0,C 180,E1 -10724.406,E2 -10724.406} C_VEL
LIN {X 0,Y 404.97,Z 146.758,A -85,B 0,C 180,E1 -10725.861,E2 -10725.861} C_VEL
LIN {X 0,Y 404.222,Z 143.136,A -85,B 0,C 180,E1 -10726.793,E2 -10726.793} C_VEL
LIN {X 0,Y 404.164,Z 143.144,A -85,B 0,C 180,E1 -10730.35,E2 -10730.35} C_VEL
LIN {X 0,Y 404.163,Z 143.138,A -85,B 0,C 180,E1 -10733.574,E2 -10733.574} C_VEL
LIN {X 0,Y 404.182,Z 143.137,A -85,B 0,C 180,E1 -10735.765,E2 -10735.765} C_VEL
LIN {X 0,Y 404.194,Z 143.138,A -85,B 0,C 180,E1 -10737.998,E2 -10737.998} C_VEL
LIN {X 0,Y 404.137,Z 143.142,A -85,B 0,C 180,E1 -10741.557,E2 -10741.557} C_VEL
LIN {X 0,Y 404.181,Z 143.136,A -85,B 0,C 180,E1 -10745.015,E2 -10745.015} C_VEL
LIN {X 0,Y 404.153,Z 143.14,A -85,B 0,C 180,E1 -10748.755,E2 -10748.755} C_VEL
LIN {X 0,Y 404.118,Z 143.147,A -85,B 0,C 180,E1 -10751.598,E2 -10751.598} C_VEL
LIN {X 0,Y 404.139,Z 143.142,A -85,B 0,C 180,E1 -10754.521,E2 -10754.521} C_VEL
LIN {X 0,Y 404.13,Z 143.144,A -85,B 0,C 180,E1 -10757.294,E2 -10757.294} C_VEL
LIN {X 0,Y 404.162,Z 143.142,A -85,B 0,C 180,E1 -10759.954,E2 -10759.954} C_VEL
LIN {X 0,Y 404.128,Z 143.144,A -85,B 0,C 180,E1 -10763.124,E2 -10763.124} C_VEL
LIN {X 0,Y 404.136,Z 143.144,A -85,B 0,C 180,E1 -10766.187,E2 -10766.187} C_VEL
LIN {X 0,Y 404.136,Z 143.145,A -85,B 0,C 180,E1 -10769.714,E2 -10769.714} C_VEL
LIN {X 0,Y 404.183,Z 143.138,A -85,B 0,C 180,E1 -10773.122,E2 -10773.122} C_VEL
LIN {X 0,Y 404.149,Z 143.14,A -85,B 0,C 180,E1 -10776.424,E2 -10776.424} C_VEL
LIN {X 0,Y 404.181,Z 143.139,A -85,B 0,C 180,E1 -10779.874,E2 -10779.874} C_VEL
LIN {X 0,Y 404.205,Z 143.136,A -85,B 0,C 180,E1 -10782.993,E2 -10782.993} C_VEL
LIN {X 0,Y 404.272,Z 143.128,A -85,B 0,C 180,E1 -10786.938,E2 -10786.938} C_VEL
LIN {X 0,Y 404.243,Z 143.129,A -85,B 0,C 180,E1 -10789.988,E2 -10789.988} C_VEL
LIN {X 0,Y 404.329,Z 143.122,A -85,B 0,C 180,E1 -10793.011,E2 -10793.011} C_VEL
LIN {X 0,Y 404.245,Z 143.132,A -85,B 0,C 180,E1 -10795.013,E2 -10795.013} C_VEL
LIN {X 0,Y 404.458,Z 143.102,A -85,B 0,C 180,E1 -10798.008,E2 -10798.008} C_VEL
LIN {X 0,Y 404.334,Z 143.121,A -85,B 0,C 180,E1 -10800.996,E2 -10800.996} C_VEL
LIN {X 0,Y 404.376,Z 143.116,A -85,B 0,C 180,E1 -10802.989,E2 -10802.989} C_VEL
LIN {X 0,Y 404.366,Z 143.113,A -85,B 0,C 180,E1 -10805.986,E2 -10805.986} C_VEL
LIN {X 0,Y 404.253,Z 143.131,A -85,B 0,C 180,E1 -10809.002,E2 -10809.002} C_VEL
LIN {X 0,Y 404.243,Z 143.129,A -85,B 0,C 180,E1 -10812.042,E2 -10812.042} C_VEL
LIN {X 0,Y 404.192,Z 143.138,A -85,B 0,C 180,E1 -10815.118,E2 -10815.118} C_VEL
LIN {X 0,Y 404.192,Z 143.137,A -85,B 0,C 180,E1 -10818.239,E2 -10818.239} C_VEL
LIN {X 0,Y 404.127,Z 143.143,A -85,B 0,C 180,E1 -10821.42,E2 -10821.42} C_VEL
LIN {X 0,Y 404.154,Z 143.144,A -85,B 0,C 180,E1 -10824.667,E2 -10824.667} C_VEL
LIN {X 0,Y 404.185,Z 143.137,A -85,B 0,C 180,E1 -10828,E2 -10828} C_VEL
LIN {X 0,Y 404.129,Z 143.143,A -85,B 0,C 180,E1 -10831.559,E2 -10831.559} C_VEL
LIN {X 0,Y 404.174,Z 143.138,A -85,B 0,C 180,E1 -10835.017,E2 -10835.017} C_VEL
LIN {X 0,Y 404.142,Z 143.143,A -85,B 0,C 180,E1 -10838.758,E2 -10838.758} C_VEL
LIN {X 0,Y 404.115,Z 143.145,A -85,B 0,C 180,E1 -10841.601,E2 -10841.601} C_VEL
LIN {X 0,Y 404.138,Z 143.144,A -85,B 0,C 180,E1 -10844.523,E2 -10844.523} C_VEL
LIN {X 0,Y 404.13,Z 143.142,A -85,B 0,C 180,E1 -10847.297,E2 -10847.297} C_VEL
LIN {X 0,Y 404.163,Z 143.142,A -85,B 0,C 180,E1 -10849.957,E2 -10849.957} C_VEL
LIN {X 0,Y 404.131,Z 143.141,A -85,B 0,C 180,E1 -10853.126,E2 -10853.126} C_VEL
LIN {X 0,Y 404.141,Z 143.145,A -85,B 0,C 180,E1 -10856.189,E2 -10856.189} C_VEL
LIN {X 0,Y 404.142,Z 143.144,A -85,B 0,C 180,E1 -10859.716,E2 -10859.716} C_VEL
LIN {X 0,Y 404.245,Z 143.188,A -85,B 0,C 180,E1 -10861.794,E2 -10861.794} C_VEL
LIN {X 0,Y 406.889,Z 156.791,A -85,B 0,C 180,E1 -10864.693,E2 -10864.693} C_VEL
LIN {X 0,Y 407.11,Z 160.917,A -85,B 0,C 180,E1 -10865.525,E2 -10865.525} C_VEL
LIN {X 0,Y 405.995,Z 177.219,A -85,B 0,C 180,E1 -10868.685,E2 -10868.685} C_VEL
LIN {X 0,Y 405.405,Z 187.251,A -85,B 0,C 180,E1 -10870.616,E2 -10870.616} C_VEL
LIN {X 0,Y 409.475,Z 217.13,A -85,B 0,C 180,E1 -10871.33,E2 -10871.33} C_VEL
LIN {X 0,Y 408.613,Z 296.404,A -85,B 0,C 180,E1 -10872.742,E2 -10872.742} C_VEL
LIN {X 0,Y 407.965,Z 310.322,A -85,B 0,C 180,E1 -10873.198,E2 -10873.198} C_VEL
LIN {X 0,Y 407.333,Z 322.252,A -85,B 0,C 180,E1 -10873.783,E2 -10873.783} C_VEL
LIN {X 0,Y 406.619,Z 334.33,A -85,B 0,C 180,E1 -10874.59,E2 -10874.59} C_VEL
LIN {X 0,Y 405.808,Z 345.87,A -85,B 0,C 180,E1 -10875.586,E2 -10875.586} C_VEL
LIN {X 0,Y 405.097,Z 356.76,A -85,B 0,C 180,E1 -10876.771,E2 -10876.771} C_VEL
LIN {X 0,Y 404.472,Z 365.614,A -85,B 0,C 180,E1 -10877.966,E2 -10877.966} C_VEL
LIN {X 0,Y 403.752,Z 374.667,A -85,B 0,C 180,E1 -10879.47,E2 -10879.47} C_VEL
LIN {X 0,Y 403.336,Z 381.964,A -85,B 0,C 180,E1 -10880.979,E2 -10880.979} C_VEL
LIN {X 0,Y 403.098,Z 387.795,A -85,B 0,C 180,E1 -10882.487,E2 -10882.487} C_VEL
LIN {X 0,Y 402.938,Z 392.379,A -85,B 0,C 180,E1 -10883.994,E2 -10883.994} C_VEL
LIN {X 0,Y 402.949,Z 394.795,A -85,B 0,C 180,E1 -10884.998,E2 -10884.998} C_VEL
LIN {X 0,Y 402.878,Z 396.77,A -85,B 0,C 180,E1 -10886,E2 -10886} C_VEL
LIN {X 0,Y 402.91,Z 398.331,A -85,B 0,C 180,E1 -10887.001,E2 -10887.001} C_VEL
LIN {X 0,Y 402.952,Z 399.442,A -85,B 0,C 180,E1 -10888.002,E2 -10888.002} C_VEL
LIN {X 0,Y 402.9,Z 400.444,A -85,B 0,C 180,E1 -10890.001,E2 -10890.001} C_VEL
LIN {X 0,Y 402.907,Z 400.365,A -85,B 0,C 180,E1 -10891,E2 -10891} C_VEL
LIN {X 0,Y 402.947,Z 399.866,A -85,B 0,C 180,E1 -10892,E2 -10892} C_VEL
LIN {X 0,Y 402.858,Z 397.636,A -85,B 0,C 180,E1 -10894.002,E2 -10894.002} C_VEL
LIN {X 0,Y 402.88,Z 394.867,A -85,B 0,C 180,E1 -10895.507,E2 -10895.507} C_VEL
LIN {X 0,Y 403.005,Z 391.082,A -85,B 0,C 180,E1 -10897.013,E2 -10897.013} C_VEL
LIN {X 0,Y 403.313,Z 386.184,A -85,B 0,C 180,E1 -10898.519,E2 -10898.519} C_VEL
LIN {X 0,Y 403.729,Z 380.027,A -85,B 0,C 180,E1 -10900.026,E2 -10900.026} C_VEL
LIN {X 0,Y 404.347,Z 372.391,A -85,B 0,C 180,E1 -10901.531,E2 -10901.531} C_VEL
LIN {X 0,Y 405.093,Z 364.597,A -85,B 0,C 180,E1 -10902.78,E2 -10902.78} C_VEL
LIN {X 0,Y 405.88,Z 354.107,A -85,B 0,C 180,E1 -10904.148,E2 -10904.148} C_VEL
LIN {X 0,Y 406.861,Z 343.288,A -85,B 0,C 180,E1 -10905.274,E2 -10905.274} C_VEL
LIN {X 0,Y 407.742,Z 332.885,A -85,B 0,C 180,E1 -10906.138,E2 -10906.138} C_VEL
LIN {X 0,Y 408.609,Z 320.402,A -85,B 0,C 180,E1 -10906.938,E2 -10906.938} C_VEL
LIN {X 0,Y 409.367,Z 308.01,A -85,B 0,C 180,E1 -10907.517,E2 -10907.517} C_VEL
LIN {X 0,Y 409.98,Z 295.421,A -85,B 0,C 180,E1 -10907.909,E2 -10907.909} C_VEL
LIN {X 0,Y 410.928,Z 216.518,A -85,B 0,C 180,E1 -10909.323,E2 -10909.323} C_VEL
LIN {X 0,Y 407.286,Z 193.697,A -85,B 0,C 180,E1 -10909.941,E2 -10909.941} C_VEL
LIN {X 0,Y 406.081,Z 186.96,A -85,B 0,C 180,E1 -10910.143,E2 -10910.143} C_VEL
LIN {X 0,Y 407.596,Z 166.831,A -85,B 0,C 180,E1 -10914.099,E2 -10914.099} C_VEL
LIN {X 0,Y 407.903,Z 161.129,A -85,B 0,C 180,E1 -10915.242,E2 -10915.242} C_VEL
LIN {X 0,Y 405.74,Z 149.964,A -85,B 0,C 180,E1 -10917.697,E2 -10917.697} C_VEL
LIN {X 0,Y 404.2,Z 143.142,A -85,B 0,C 180,E1 -10919.28,E2 -10919.28} C_VEL
LIN {X 0,Y 404.144,Z 143.146,A -85,B 0,C 180,E1 -10922.622,E2 -10922.622} C_VEL
LIN {X 0,Y 404.183,Z 143.136,A -85,B 0,C 180,E1 -10925.19,E2 -10925.19} C_VEL
LIN {X 0,Y 404.15,Z 143.138,A -85,B 0,C 180,E1 -10928.758,E2 -10928.758} C_VEL
LIN {X 0,Y 404.121,Z 143.147,A -85,B 0,C 180,E1 -10931.599,E2 -10931.599} C_VEL
LIN {X 0,Y 404.147,Z 143.14,A -85,B 0,C 180,E1 -10934.522,E2 -10934.522} C_VEL
LIN {X 0,Y 404.133,Z 143.146,A -85,B 0,C 180,E1 -10937.295,E2 -10937.295} C_VEL
LIN {X 0,Y 404.134,Z 143.143,A -85,B 0,C 180,E1 -10939.951,E2 -10939.951} C_VEL
LIN {X 0,Y 404.136,Z 143.146,A -85,B 0,C 180,E1 -10943.126,E2 -10943.126} C_VEL
LIN {X 0,Y 404.139,Z 143.142,A -85,B 0,C 180,E1 -10946.187,E2 -10946.187} C_VEL
LIN {X 0,Y 404.145,Z 143.141,A -85,B 0,C 180,E1 -10949.715,E2 -10949.715} C_VEL
LIN {X 0,Y 404.125,Z 143.145,A -85,B 0,C 180,E1 -10953.118,E2 -10953.118} C_VEL
LIN {X 0,Y 404.15,Z 143.143,A -85,B 0,C 180,E1 -10956.424,E2 -10956.424} C_VEL
LIN {X 0,Y 404.156,Z 143.135,A -85,B 0,C 180,E1 -10959.888,E2 -10959.888} C_VEL
LIN {X 0,Y 404.174,Z 143.138,A -85,B 0,C 180,E1 -10963.013,E2 -10963.013} C_VEL
LIN {X 0,Y 404.284,Z 143.122,A -85,B 0,C 180,E1 -10966.939,E2 -10966.939} C_VEL
LIN {X 0,Y 404.24,Z 143.132,A -85,B 0,C 180,E1 -10969.988,E2 -10969.988} C_VEL
LIN {X 0,Y 404.34,Z 143.114,A -85,B 0,C 180,E1 -10973.012,E2 -10973.012} C_VEL
LIN {X 0,Y 404.253,Z 143.126,A -85,B 0,C 180,E1 -10975.013,E2 -10975.013} C_VEL
LIN {X 0,Y 404.469,Z 143.097,A -85,B 0,C 180,E1 -10978.009,E2 -10978.009} C_VEL
LIN {X 0,Y 404.346,Z 143.115,A -85,B 0,C 180,E1 -10980.996,E2 -10980.996} C_VEL
LIN {X 0,Y 404.361,Z 143.105,A -85,B 0,C 180,E1 -10982.989,E2 -10982.989} C_VEL
LIN {X 0,Y 404.343,Z 143.115,A -85,B 0,C 180,E1 -10986.47,E2 -10986.47} C_VEL
LIN {X 0,Y 404.265,Z 143.118,A -85,B 0,C 180,E1 -10989.002,E2 -10989.002} C_VEL
LIN {X 0,Y 404.256,Z 143.127,A -85,B 0,C 180,E1 -10992.042,E2 -10992.042} C_VEL
LIN {X 0,Y 404.204,Z 143.129,A -85,B 0,C 180,E1 -10995.118,E2 -10995.118} C_VEL
LIN {X 0,Y 404.205,Z 143.131,A -85,B 0,C 180,E1 -10998.239,E2 -10998.239} C_VEL
LIN {X 0,Y 404.139,Z 143.145,A -85,B 0,C 180,E1 -11001.42,E2 -11001.42} C_VEL
LIN {X 0,Y 404.162,Z 143.135,A -85,B 0,C 180,E1 -11004.667,E2 -11004.667} C_VEL
LIN {X 0,Y 404.169,Z 143.135,A -85,B 0,C 180,E1 -11008.002,E2 -11008.002} C_VEL
LIN {X 0,Y 404.141,Z 143.14,A -85,B 0,C 180,E1 -11011.558,E2 -11011.558} C_VEL
LIN {X 0,Y 404.186,Z 143.137,A -85,B 0,C 180,E1 -11015.016,E2 -11015.016} C_VEL
LIN {X 0,Y 404.151,Z 143.14,A -85,B 0,C 180,E1 -11018.758,E2 -11018.758} C_VEL
LIN {X 0,Y 404.125,Z 143.131,A -85,B 0,C 180,E1 -11021.6,E2 -11021.6} C_VEL
LIN {X 0,Y 404.148,Z 143.143,A -85,B 0,C 180,E1 -11024.522,E2 -11024.522} C_VEL
LIN {X 0,Y 404.136,Z 143.141,A -85,B 0,C 180,E1 -11027.295,E2 -11027.295} C_VEL
LIN {X 0,Y 404.157,Z 143.142,A -85,B 0,C 180,E1 -11029.953,E2 -11029.953} C_VEL
LIN {X 0,Y 404.139,Z 143.142,A -85,B 0,C 180,E1 -11033.125,E2 -11033.125} C_VEL
LIN {X 0,Y 404.149,Z 143.144,A -85,B 0,C 180,E1 -11036.188,E2 -11036.188} C_VEL
LIN {X 0,Y 404.15,Z 143.145,A -85,B 0,C 180,E1 -11039.715,E2 -11039.715} C_VEL
LIN {X 0,Y 404.204,Z 143.156,A -85,B 0,C 180,E1 -11042.389,E2 -11042.389} C_VEL
LIN {X 0,Y 406.279,Z 153.244,A -85,B 0,C 180,E1 -11044.926,E2 -11044.926} C_VEL
LIN {X 0,Y 409.308,Z 163.478,A -85,B 0,C 180,E1 -11045.289,E2 -11045.289} C_VEL
LIN {X 0,Y 411.592,Z 174.211,A -85,B 0,C 180,E1 -11045.614,E2 -11045.614} C_VEL
LIN {X 0,Y 410.349,Z 260.934,A -85,B 0,C 180,E1 -11047.167,E2 -11047.167} C_VEL
LIN {X 0,Y 409.81,Z 274.865,A -85,B 0,C 180,E1 -11047.635,E2 -11047.635} C_VEL
LIN {X 0,Y 409.229,Z 287.273,A -85,B 0,C 180,E1 -11048.262,E2 -11048.262} C_VEL
LIN {X 0,Y 408.513,Z 299.205,A -85,B 0,C 180,E1 -11049.085,E2 -11049.085} C_VEL
LIN {X 0,Y 407.577,Z 310.605,A -85,B 0,C 180,E1 -11050.089,E2 -11050.089} C_VEL
LIN {X 0,Y 406.736,Z 320.839,A -85,B 0,C 180,E1 -11051.226,E2 -11051.226} C_VEL
LIN {X 0,Y 405.974,Z 330.25,A -85,B 0,C 180,E1 -11052.533,E2 -11052.533} C_VEL
LIN {X 0,Y 405.186,Z 338.231,A -85,B 0,C 180,E1 -11053.887,E2 -11053.887} C_VEL
LIN {X 0,Y 404.486,Z 345.488,A -85,B 0,C 180,E1 -11055.407,E2 -11055.407} C_VEL
LIN {X 0,Y 403.915,Z 351.525,A -85,B 0,C 180,E1 -11057.005,E2 -11057.005} C_VEL
LIN {X 0,Y 403.553,Z 355.797,A -85,B 0,C 180,E1 -11058.446,E2 -11058.446} C_VEL
LIN {X 0,Y 403.211,Z 359.228,A -85,B 0,C 180,E1 -11059.961,E2 -11059.961} C_VEL
LIN {X 0,Y 403.129,Z 360.929,A -85,B 0,C 180,E1 -11060.972,E2 -11060.972} C_VEL
LIN {X 0,Y 403.058,Z 363.12,A -85,B 0,C 180,E1 -11062.988,E2 -11062.988} C_VEL
LIN {X 0,Y 403.01,Z 363.621,A -85,B 0,C 180,E1 -11063.993,E2 -11063.993} C_VEL
LIN {X 0,Y 402.994,Z 363.696,A -85,B 0,C 180,E1 -11064.997,E2 -11064.997} C_VEL
LIN {X 0,Y 403.004,Z 362.708,A -85,B 0,C 180,E1 -11067,E2 -11067} C_VEL
LIN {X 0,Y 403.004,Z 361.632,A -85,B 0,C 180,E1 -11068,E2 -11068} C_VEL
LIN {X 0,Y 402.993,Z 360.115,A -85,B 0,C 180,E1 -11069,E2 -11069} C_VEL
LIN {X 0,Y 403.181,Z 357.166,A -85,B 0,C 180,E1 -11070.453,E2 -11070.453} C_VEL
LIN {X 0,Y 402.654,Z 355.27,A -85,B 0,C 180,E1 -11071.245,E2 -11071.245} C_VEL
LIN {X 0,Y 400.014,Z 351.709,A -85,B 0,C 180,E1 -11072.512,E2 -11072.512} C_VEL
LIN {X 0,Y 397.436,Z 347.456,A -85,B 0,C 180,E1 -11073.75,E2 -11073.75} C_VEL
LIN {X 0,Y 397.018,Z 344.453,A -85,B 0,C 180,E1 -11074.485,E2 -11074.485} C_VEL
LIN {X 0,Y 397.675,Z 336.584,A -85,B 0,C 180,E1 -11076.086,E2 -11076.086} C_VEL
LIN {X 0,Y 398.351,Z 328.899,A -85,B 0,C 180,E1 -11077.348,E2 -11077.348} C_VEL
LIN {X 0,Y 399.215,Z 318.463,A -85,B 0,C 180,E1 -11078.732,E2 -11078.732} C_VEL
LIN {X 0,Y 400.012,Z 307.845,A -85,B 0,C 180,E1 -11079.862,E2 -11079.862} C_VEL
LIN {X 0,Y 400.689,Z 296.543,A -85,B 0,C 180,E1 -11080.816,E2 -11080.816} C_VEL
LIN {X 0,Y 401.258,Z 284.138,A -85,B 0,C 180,E1 -11081.619,E2 -11081.619} C_VEL
LIN {X 0,Y 401.765,Z 271.516,A -85,B 0,C 180,E1 -11082.212,E2 -11082.212} C_VEL
LIN {X 0,Y 402.054,Z 259.451,A -85,B 0,C 180,E1 -11082.588,E2 -11082.588} C_VEL
LIN {X 0,Y 403.083,Z 173.712,A -85,B 0,C 180,E1 -11084.127,E2 -11084.127} C_VEL
LIN {X 0,Y 398.946,Z 153.177,A -85,B 0,C 180,E1 -11084.722,E2 -11084.722} C_VEL
LIN {X 0,Y 397.172,Z 144.014,A -85,B 0,C 180,E1 -11087.004,E2 -11087.004} C_VEL
LIN {X 0,Y 397.139,Z 144.019,A -85,B 0,C 180,E1 -11090.294,E2 -11090.294} C_VEL
LIN {X 0,Y 397.128,Z 144.017,A -85,B 0,C 180,E1 -11094.017,E2 -11094.017} C_VEL
LIN {X 0,Y 397.193,Z 144.006,A -85,B 0,C 180,E1 -11097.389,E2 -11097.389} C_VEL
LIN {X 0,Y 397.076,Z 144.021,A -85,B 0,C 180,E1 -11100.881,E2 -11100.881} C_VEL
LIN {X 0,Y 397.122,Z 144.017,A -85,B 0,C 180,E1 -11104.492,E2 -11104.492} C_VEL
LIN {X 0,Y 397.1,Z 144.021,A -85,B 0,C 180,E1 -11108.273,E2 -11108.273} C_VEL
LIN {X 0,Y 397.084,Z 144.02,A -85,B 0,C 180,E1 -11110.907,E2 -11110.907} C_VEL
LIN {X 0,Y 397.096,Z 144.022,A -85,B 0,C 180,E1 -11113.647,E2 -11113.647} C_VEL
LIN {X 0,Y 397.096,Z 144.019,A -85,B 0,C 180,E1 -11116.52,E2 -11116.52} C_VEL
LIN {X 0,Y 397.105,Z 144.018,A -85,B 0,C 180,E1 -11120.421,E2 -11120.421} C_VEL
LIN {X 0,Y 397.1,Z 144.02,A -85,B 0,C 180,E1 -11124.264,E2 -11124.264} C_VEL
LIN {X 0,Y 397.106,Z 144.017,A -85,B 0,C 180,E1 -11126.726,E2 -11126.726} C_VEL
LIN {X 0,Y 397.115,Z 144.017,A -85,B 0,C 180,E1 -11130.295,E2 -11130.295} C_VEL
LIN {X 0,Y 397.184,Z 144.008,A -85,B 0,C 180,E1 -11132.609,E2 -11132.609} C_VEL
LIN {X 0,Y 397.113,Z 144.019,A -85,B 0,C 180,E1 -11135.98,E2 -11135.98} C_VEL
LIN {X 0,Y 397.128,Z 144.018,A -85,B 0,C 180,E1 -11139.704,E2 -11139.704} C_VEL
LIN {X 0,Y 397.171,Z 144.011,A -85,B 0,C 180,E1 -11142.844,E2 -11142.844} C_VEL
LIN {X 0,Y 397.218,Z 144.005,A -85,B 0,C 180,E1 -11146.702,E2 -11146.702} C_VEL
LIN {X 0,Y 397.203,Z 144.007,A -85,B 0,C 180,E1 -11149.808,E2 -11149.808} C_VEL
LIN {X 0,Y 397.281,Z 143.999,A -85,B 0,C 180,E1 -11152.887,E2 -11152.887} C_VEL
LIN {X 0,Y 397.216,Z 144.008,A -85,B 0,C 180,E1 -11154.925,E2 -11154.925} C_VEL
LIN {X 0,Y 397.427,Z 143.978,A -85,B 0,C 180,E1 -11157.973,E2 -11157.973} C_VEL
LIN {X 0,Y 397.427,Z 143.978,A -85,B 0,C 180,E1 -11162.027,E2 -11162.027} C_VEL
LIN {X 0,Y 397.318,Z 143.991,A -85,B 0,C 180,E1 -11166.092,E2 -11166.092} C_VEL
LIN {X 0,Y 397.223,Z 144.007,A -85,B 0,C 180,E1 -11169.162,E2 -11169.162} C_VEL
LIN {X 0,Y 397.207,Z 144.006,A -85,B 0,C 180,E1 -11172.258,E2 -11172.258} C_VEL
LIN {X 0,Y 397.165,Z 144.011,A -85,B 0,C 180,E1 -11175.393,E2 -11175.393} C_VEL
LIN {X 0,Y 397.146,Z 144.016,A -85,B 0,C 180,E1 -11178.574,E2 -11178.574} C_VEL
LIN {X 0,Y 397.084,Z 144.02,A -85,B 0,C 180,E1 -11181.819,E2 -11181.819} C_VEL
LIN {X 0,Y 397.116,Z 144.018,A -85,B 0,C 180,E1 -11185.134,E2 -11185.134} C_VEL
LIN {X 0,Y 397.152,Z 144.012,A -85,B 0,C 180,E1 -11187.777,E2 -11187.777} C_VEL
LIN {X 0,Y 397.069,Z 144.024,A -85,B 0,C 180,E1 -11190.883,E2 -11190.883} C_VEL
LIN {X 0,Y 397.116,Z 144.021,A -85,B 0,C 180,E1 -11194.494,E2 -11194.494} C_VEL
LIN {X 0,Y 397.091,Z 144.023,A -85,B 0,C 180,E1 -11198.276,E2 -11198.276} C_VEL
LIN {X 0,Y 397.081,Z 144.021,A -85,B 0,C 180,E1 -11200.91,E2 -11200.91} C_VEL
LIN {X 0,Y 397.094,Z 144.02,A -85,B 0,C 180,E1 -11203.65,E2 -11203.65} C_VEL
LIN {X 0,Y 397.096,Z 144.021,A -85,B 0,C 180,E1 -11206.522,E2 -11206.522} C_VEL
LIN {X 0,Y 397.109,Z 144.02,A -85,B 0,C 180,E1 -11210.424,E2 -11210.424} C_VEL
LIN {X 0,Y 397.103,Z 144.021,A -85,B 0,C 180,E1 -11214.267,E2 -11214.267} C_VEL
LIN {X 0,Y 397.11,Z 144.016,A -85,B 0,C 180,E1 -11216.728,E2 -11216.728} C_VEL
LIN {X 0,Y 397.121,Z 144.021,A -85,B 0,C 180,E1 -11220.297,E2 -11220.297} C_VEL
LIN {X 0,Y 397.217,Z 144.175,A -85,B 0,C 180,E1 -11221.567,E2 -11221.567} C_VEL
LIN {X 0,Y 399.88,Z 157.639,A -85,B 0,C 180,E1 -11224.496,E2 -11224.496} C_VEL
LIN {X 0,Y 400.164,Z 161.908,A -85,B 0,C 180,E1 -11225.376,E2 -11225.376} C_VEL
LIN {X 0,Y 398.913,Z 179.053,A -85,B 0,C 180,E1 -11228.756,E2 -11228.756} C_VEL
LIN {X 0,Y 398.49,Z 186.867,A -85,B 0,C 180,E1 -11230.289,E2 -11230.289} C_VEL
LIN {X 0,Y 402.669,Z 217.589,A -85,B 0,C 180,E1 -11231.05,E2 -11231.05} C_VEL
LIN {X 0,Y 401.775,Z 296.083,A -85,B 0,C 180,E1 -11232.472,E2 -11232.472} C_VEL
LIN {X 0,Y 401.122,Z 310.003,A -85,B 0,C 180,E1 -11232.935,E2 -11232.935} C_VEL
LIN {X 0,Y 400.429,Z 322.474,A -85,B 0,C 180,E1 -11233.561,E2 -11233.561} C_VEL
LIN {X 0,Y 399.618,Z 335.204,A -85,B 0,C 180,E1 -11234.444,E2 -11234.444} C_VEL
LIN {X 0,Y 398.783,Z 346.524,A -85,B 0,C 180,E1 -11235.456,E2 -11235.456} C_VEL
LIN {X 0,Y 398.135,Z 356.41,A -85,B 0,C 180,E1 -11236.564,E2 -11236.564} C_VEL
LIN {X 0,Y 397.475,Z 365.086,A -85,B 0,C 180,E1 -11237.751,E2 -11237.751} C_VEL
LIN {X 0,Y 396.742,Z 374.175,A -85,B 0,C 180,E1 -11239.282,E2 -11239.282} C_VEL
LIN {X 0,Y 396.298,Z 381.503,A -85,B 0,C 180,E1 -11240.817,E2 -11240.817} C_VEL
LIN {X 0,Y 396.03,Z 387.367,A -85,B 0,C 180,E1 -11242.353,E2 -11242.353} C_VEL
LIN {X 0,Y 395.827,Z 392.741,A -85,B 0,C 180,E1 -11244.195,E2 -11244.195} C_VEL
LIN {X 0,Y 395.799,Z 396.392,A -85,B 0,C 180,E1 -11245.928,E2 -11245.928} C_VEL
LIN {X 0,Y 395.81,Z 397.963,A -85,B 0,C 180,E1 -11246.948,E2 -11246.948} C_VEL
LIN {X 0,Y 395.883,Z 399.096,A -85,B 0,C 180,E1 -11247.966,E2 -11247.966} C_VEL
LIN {X 0,Y 395.825,Z 400.116,A -85,B 0,C 180,E1 -11250.001,E2 -11250.001} C_VEL
LIN {X 0,Y 395.834,Z 400.046,A -85,B 0,C 180,E1 -11251.018,E2 -11251.018} C_VEL
LIN {X 0,Y 395.858,Z 399.566,A -85,B 0,C 180,E1 -11252.036,E2 -11252.036} C_VEL
LIN {X 0,Y 395.779,Z 397.355,A -85,B 0,C 180,E1 -11254.074,E2 -11254.074} C_VEL
LIN {X 0,Y 395.786,Z 394.306,A -85,B 0,C 180,E1 -11255.748,E2 -11255.748} C_VEL
LIN {X 0,Y 396.053,Z 389.367,A -85,B 0,C 180,E1 -11257.649,E2 -11257.649} C_VEL
LIN {X 0,Y 396.436,Z 383.072,A -85,B 0,C 180,E1 -11259.439,E2 -11259.439} C_VEL
LIN {X 0,Y 396.964,Z 376.237,A -85,B 0,C 180,E1 -11260.972,E2 -11260.972} C_VEL
LIN {X 0,Y 397.87,Z 367.75,A -85,B 0,C 180,E1 -11262.498,E2 -11262.498} C_VEL
LIN {X 0,Y 398.591,Z 358.379,A -85,B 0,C 180,E1 -11263.858,E2 -11263.858} C_VEL
LIN {X 0,Y 399.623,Z 347.262,A -85,B 0,C 180,E1 -11265.153,E2 -11265.153} C_VEL
LIN {X 0,Y 400.647,Z 336.127,A -85,B 0,C 180,E1 -11266.17,E2 -11266.17} C_VEL
LIN {X 0,Y 401.646,Z 323.802,A -85,B 0,C 180,E1 -11267.044,E2 -11267.044} C_VEL
LIN {X 0,Y 402.482,Z 312.131,A -85,B 0,C 180,E1 -11267.662,E2 -11267.662} C_VEL
LIN {X 0,Y 403.152,Z 299.658,A -85,B 0,C 180,E1 -11268.124,E2 -11268.124} C_VEL
LIN {X 0,Y 403.522,Z 282.691,A -85,B 0,C 180,E1 -11268.489,E2 -11268.489} C_VEL
LIN {X 0,Y 404.222,Z 216.728,A -85,B 0,C 180,E1 -11269.68,E2 -11269.68} C_VEL
LIN {X 0,Y 400.551,Z 194.038,A -85,B 0,C 180,E1 -11270.313,E2 -11270.313} C_VEL
LIN {X 0,Y 399.215,Z 186.515,A -85,B 0,C 180,E1 -11270.562,E2 -11270.562} C_VEL
LIN {X 0,Y 400.761,Z 167.056,A -85,B 0,C 180,E1 -11274.459,E2 -11274.459} C_VEL
LIN {X 0,Y 400.968,Z 162.311,A -85,B 0,C 180,E1 -11275.432,E2 -11275.432} C_VEL
LIN {X 0,Y 398.558,Z 150.211,A -85,B 0,C 180,E1 -11278.154,E2 -11278.154} C_VEL
LIN {X 0,Y 397.123,Z 144.025,A -85,B 0,C 180,E1 -11279.632,E2 -11279.632} C_VEL
LIN {X 0,Y 397.117,Z 144.02,A -85,B 0,C 180,E1 -11283.273,E2 -11283.273} C_VEL
LIN {X 0,Y 397.11,Z 144.023,A -85,B 0,C 180,E1 -11285.735,E2 -11285.735} C_VEL
LIN {X 0,Y 397.105,Z 144.017,A -85,B 0,C 180,E1 -11289.579,E2 -11289.579} C_VEL
LIN {X 0,Y 397.103,Z 144.022,A -85,B 0,C 180,E1 -11293.479,E2 -11293.479} C_VEL
LIN {X 0,Y 397.102,Z 144.019,A -85,B 0,C 180,E1 -11296.521,E2 -11296.521} C_VEL
LIN {X 0,Y 397.088,Z 144.021,A -85,B 0,C 180,E1 -11300.42,E2 -11300.42} C_VEL
LIN {X 0,Y 397.098,Z 144.023,A -85,B 0,C 180,E1 -11303.005,E2 -11303.005} C_VEL
LIN {X 0,Y 397.113,Z 144.021,A -85,B 0,C 180,E1 -11306.727,E2 -11306.727} C_VEL
LIN {X 0,Y 397.118,Z 144.017,A -85,B 0,C 180,E1 -11310.295,E2 -11310.295} C_VEL
LIN {X 0,Y 397.087,Z 144.019,A -85,B 0,C 180,E1 -11313.738,E2 -11313.738} C_VEL
LIN {X 0,Y 397.1,Z 144.02,A -85,B 0,C 180,E1 -11317.085,E2 -11317.085} C_VEL
LIN {X 0,Y 397.131,Z 144.01,A -85,B 0,C 180,E1 -11320.352,E2 -11320.352} C_VEL
LIN {X 0,Y 397.128,Z 144.014,A -85,B 0,C 180,E1 -11323.552,E2 -11323.552} C_VEL
LIN {X 0,Y 397.23,Z 144.001,A -85,B 0,C 180,E1 -11326.703,E2 -11326.703} C_VEL
LIN {X 0,Y 397.202,Z 144.007,A -85,B 0,C 180,E1 -11329.809,E2 -11329.809} C_VEL
LIN {X 0,Y 397.293,Z 143.993,A -85,B 0,C 180,E1 -11332.887,E2 -11332.887} C_VEL
LIN {X 0,Y 397.225,Z 144.002,A -85,B 0,C 180,E1 -11334.925,E2 -11334.925} C_VEL
LIN {X 0,Y 397.436,Z 143.973,A -85,B 0,C 180,E1 -11337.973,E2 -11337.973} C_VEL
LIN {X 0,Y 397.317,Z 143.99,A -85,B 0,C 180,E1 -11341.014,E2 -11341.014} C_VEL
LIN {X 0,Y 397.297,Z 143.985,A -85,B 0,C 180,E1 -11343.042,E2 -11343.042} C_VEL
LIN {X 0,Y 397.3,Z 143.992,A -85,B 0,C 180,E1 -11346.463,E2 -11346.463} C_VEL
LIN {X 0,Y 397.235,Z 143.994,A -85,B 0,C 180,E1 -11349.162,E2 -11349.162} C_VEL
LIN {X 0,Y 397.219,Z 144.002,A -85,B 0,C 180,E1 -11352.258,E2 -11352.258} C_VEL
LIN {X 0,Y 397.178,Z 144.007,A -85,B 0,C 180,E1 -11355.392,E2 -11355.392} C_VEL
LIN {X 0,Y 397.159,Z 144.009,A -85,B 0,C 180,E1 -11358.574,E2 -11358.574} C_VEL
LIN {X 0,Y 397.097,Z 144.019,A -85,B 0,C 180,E1 -11361.819,E2 -11361.819} C_VEL
LIN {X 0,Y 397.109,Z 144.017,A -85,B 0,C 180,E1 -11365.135,E2 -11365.135} C_VEL
LIN {X 0,Y 397.101,Z 144.018,A -85,B 0,C 180,E1 -11368.546,E2 -11368.546} C_VEL
LIN {X 0,Y 397.08,Z 144.02,A -85,B 0,C 180,E1 -11372.072,E2 -11372.072} C_VEL
LIN {X 0,Y 397.121,Z 144.014,A -85,B 0,C 180,E1 -11375.503,E2 -11375.503} C_VEL
LIN {X 0,Y 397.128,Z 144.014,A -85,B 0,C 180,E1 -11378.86,E2 -11378.86} C_VEL
LIN {X 0,Y 397.071,Z 144.014,A -85,B 0,C 180,E1 -11382.267,E2 -11382.267} C_VEL
LIN {X 0,Y 397.09,Z 144.018,A -85,B 0,C 180,E1 -11385.069,E2 -11385.069} C_VEL
LIN {X 0,Y 397.065,Z 144.025,A -85,B 0,C 180,E1 -11388.022,E2 -11388.022} C_VEL
LIN {X 0,Y 397.128,Z 144.015,A -85,B 0,C 180,E1 -11391.14,E2 -11391.14} C_VEL
LIN {X 0,Y 397.123,Z 144.019,A -85,B 0,C 180,E1 -11394.497,E2 -11394.497} C_VEL
LIN {X 0,Y 397.083,Z 144.022,A -85,B 0,C 180,E1 -11397.928,E2 -11397.928} C_VEL
LIN {X 0,Y 397.123,Z 144.021,A -85,B 0,C 180,E1 -11401.456,E2 -11401.456} C_VEL
LIN {X 0,Y 397.174,Z 144.223,A -85,B 0,C 180,E1 -11402.114,E2 -11402.114} C_VEL
LIN {X 0,Y 399.216,Z 153.668,A -85,B 0,C 180,E1 -11404.518,E2 -11404.518} C_VEL
LIN {X 0,Y 402.484,Z 163.664,A -85,B 0,C 180,E1 -11404.902,E2 -11404.902} C_VEL
LIN {X 0,Y 404.96,Z 174.663,A -85,B 0,C 180,E1 -11405.251,E2 -11405.251} C_VEL
LIN {X 0,Y 403.736,Z 260.351,A -85,B 0,C 180,E1 -11406.806,E2 -11406.806} C_VEL
LIN {X 0,Y 403.192,Z 273.819,A -85,B 0,C 180,E1 -11407.247,E2 -11407.247} C_VEL
LIN {X 0,Y 402.578,Z 286.055,A -85,B 0,C 180,E1 -11407.851,E2 -11407.851} C_VEL
LIN {X 0,Y 401.945,Z 297.186,A -85,B 0,C 180,E1 -11408.592,E2 -11408.592} C_VEL
LIN {X 0,Y 400.99,Z 309.051,A -85,B 0,C 180,E1 -11409.613,E2 -11409.613} C_VEL
LIN {X 0,Y 400.117,Z 318.562,A -85,B 0,C 180,E1 -11410.637,E2 -11410.637} C_VEL
LIN {X 0,Y 399.311,Z 327.962,A -85,B 0,C 180,E1 -11411.883,E2 -11411.883} C_VEL
LIN {X 0,Y 398.471,Z 336.893,A -85,B 0,C 180,E1 -11413.344,E2 -11413.344} C_VEL
LIN {X 0,Y 397.64,Z 344.445,A -85,B 0,C 180,E1 -11414.888,E2 -11414.888} C_VEL
LIN {X 0,Y 396.97,Z 351.396,A -85,B 0,C 180,E1 -11416.693,E2 -11416.693} C_VEL
LIN {X 0,Y 396.529,Z 355.972,A -85,B 0,C 180,E1 -11418.239,E2 -11418.239} C_VEL
LIN {X 0,Y 396.165,Z 359.44,A -85,B 0,C 180,E1 -11419.781,E2 -11419.781} C_VEL
LIN {X 0,Y 396.062,Z 361.173,A -85,B 0,C 180,E1 -11420.81,E2 -11420.81} C_VEL
LIN {X 0,Y 395.979,Z 363.4,A -85,B 0,C 180,E1 -11422.862,E2 -11422.862} C_VEL
LIN {X 0,Y 395.952,Z 363.929,A -85,B 0,C 180,E1 -11423.886,E2 -11423.886} C_VEL
LIN {X 0,Y 395.906,Z 364.029,A -85,B 0,C 180,E1 -11424.907,E2 -11424.907} C_VEL
LIN {X 0,Y 395.904,Z 363.077,A -85,B 0,C 180,E1 -11426.946,E2 -11426.946} C_VEL
LIN {X 0,Y 395.933,Z 362.027,A -85,B 0,C 180,E1 -11427.965,E2 -11427.965} C_VEL
LIN {X 0,Y 395.915,Z 360.538,A -85,B 0,C 180,E1 -11428.982,E2 -11428.982} C_VEL
LIN {X 0,Y 396.122,Z 357.525,A -85,B 0,C 180,E1 -11430.507,E2 -11430.507} C_VEL
LIN {X 0,Y 396.327,Z 353.482,A -85,B 0,C 180,E1 -11432.031,E2 -11432.031} C_VEL
LIN {X 0,Y 396.73,Z 348.28,A -85,B 0,C 180,E1 -11433.554,E2 -11433.554} C_VEL
LIN {X 0,Y 397.018,Z 344.453,A -85,B 0,C 180,E1 -11434.485,E2 -11434.485} C_VEL
LIN {X 0,Y 396.653,Z 341.263,A -85,B 0,C 180,E1 -11435.202,E2 -11435.202} C_VEL
LIN {X 0,Y 394.336,Z 335.765,A -85,B 0,C 180,E1 -11436.351,E2 -11436.351} C_VEL
LIN {X 0,Y 392.038,Z 329.68,A -85,B 0,C 180,E1 -11437.445,E2 -11437.445} C_VEL
LIN {X 0,Y 391.703,Z 325.569,A -85,B 0,C 180,E1 -11438.066,E2 -11438.066} C_VEL
LIN {X 0,Y 392.502,Z 316.024,A -85,B 0,C 180,E1 -11439.273,E2 -11439.273} C_VEL
LIN {X 0,Y 393.29,Z 304.462,A -85,B 0,C 180,E1 -11440.44,E2 -11440.44} C_VEL
LIN {X 0,Y 394.008,Z 293.45,A -85,B 0,C 180,E1 -11441.314,E2 -11441.314} C_VEL
LIN {X 0,Y 394.512,Z 282.076,A -85,B 0,C 180,E1 -11442.016,E2 -11442.016} C_VEL
LIN {X 0,Y 395.049,Z 269.005,A -85,B 0,C 180,E1 -11442.586,E2 -11442.586} C_VEL
LIN {X 0,Y 395.296,Z 256.454,A -85,B 0,C 180,E1 -11442.937,E2 -11442.937} C_VEL
LIN {X 0,Y 396.4,Z 175.039,A -85,B 0,C 180,E1 -11444.409,E2 -11444.409} C_VEL
LIN {X 0,Y 392.233,Z 154.841,A -85,B 0,C 180,E1 -11444.987,E2 -11444.987} C_VEL
LIN {X 0,Y 391.86,Z 153.42,A -85,B 0,C 180,E1 -11445.072,E2 -11445.072} C_VEL
LIN {X 0,Y 390.149,Z 144.888,A -85,B 0,C 180,E1 -11447.231,E2 -11447.231} C_VEL
LIN {X 0,Y 390.088,Z 144.896,A -85,B 0,C 180,E1 -11450.469,E2 -11450.469} C_VEL
LIN {X 0,Y 390.077,Z 144.896,A -85,B 0,C 180,E1 -11454.48,E2 -11454.48} C_VEL
LIN {X 0,Y 390.116,Z 144.891,A -85,B 0,C 180,E1 -11457.929,E2 -11457.929} C_VEL
LIN {X 0,Y 390.021,Z 144.9,A -85,B 0,C 180,E1 -11461.503,E2 -11461.503} C_VEL
LIN {X 0,Y 390.082,Z 144.892,A -85,B 0,C 180,E1 -11465.205,E2 -11465.205} C_VEL
LIN {X 0,Y 390.066,Z 144.894,A -85,B 0,C 180,E1 -11469.217,E2 -11469.217} C_VEL
LIN {X 0,Y 390.038,Z 144.9,A -85,B 0,C 180,E1 -11472.373,E2 -11472.373} C_VEL
LIN {X 0,Y 390.038,Z 144.899,A -85,B 0,C 180,E1 -11475.353,E2 -11475.353} C_VEL
LIN {X 0,Y 390.024,Z 144.902,A -85,B 0,C 180,E1 -11478.185,E2 -11478.185} C_VEL
LIN {X 0,Y 390.08,Z 144.892,A -85,B 0,C 180,E1 -11480.906,E2 -11480.906} C_VEL
LIN {X 0,Y 390.076,Z 144.893,A -85,B 0,C 180,E1 -11484.792,E2 -11484.792} C_VEL
LIN {X 0,Y 390.014,Z 144.901,A -85,B 0,C 180,E1 -11488.495,E2 -11488.495} C_VEL
LIN {X 0,Y 390.108,Z 144.891,A -85,B 0,C 180,E1 -11492.069,E2 -11492.069} C_VEL
LIN {X 0,Y 390.052,Z 144.9,A -85,B 0,C 180,E1 -11495.517,E2 -11495.517} C_VEL
LIN {X 0,Y 390.045,Z 144.898,A -85,B 0,C 180,E1 -11498.877,E2 -11498.877} C_VEL
LIN {X 0,Y 390.1,Z 144.89,A -85,B 0,C 180,E1 -11502.165,E2 -11502.165} C_VEL
LIN {X 0,Y 390.128,Z 144.891,A -85,B 0,C 180,E1 -11505.392,E2 -11505.392} C_VEL
LIN {X 0,Y 390.134,Z 144.887,A -85,B 0,C 180,E1 -11508.571,E2 -11508.571} C_VEL
LIN {X 0,Y 390.245,Z 144.872,A -85,B 0,C 180,E1 -11512.086,E2 -11512.086} C_VEL
LIN {X 0,Y 390.187,Z 144.883,A -85,B 0,C 180,E1 -11514.833,E2 -11514.833} C_VEL
LIN {X 0,Y 390.394,Z 144.854,A -85,B 0,C 180,E1 -11517.937,E2 -11517.937} C_VEL
LIN {X 0,Y 390.394,Z 144.853,A -85,B 0,C 180,E1 -11522.063,E2 -11522.063} C_VEL
LIN {X 0,Y 390.272,Z 144.869,A -85,B 0,C 180,E1 -11526.203,E2 -11526.203} C_VEL
LIN {X 0,Y 390.181,Z 144.882,A -85,B 0,C 180,E1 -11529.329,E2 -11529.329} C_VEL
LIN {X 0,Y 390.159,Z 144.886,A -85,B 0,C 180,E1 -11532.483,E2 -11532.483} C_VEL
LIN {X 0,Y 390.126,Z 144.887,A -85,B 0,C 180,E1 -11535.677,E2 -11535.677} C_VEL
LIN {X 0,Y 390.091,Z 144.895,A -85,B 0,C 180,E1 -11538.923,E2 -11538.923} C_VEL
LIN {X 0,Y 390.026,Z 144.902,A -85,B 0,C 180,E1 -11542.235,E2 -11542.235} C_VEL
LIN {X 0,Y 390.087,Z 144.892,A -85,B 0,C 180,E1 -11545.737,E2 -11545.737} C_VEL
LIN {X 0,Y 390.048,Z 144.897,A -85,B 0,C 180,E1 -11549.11,E2 -11549.11} C_VEL
LIN {X 0,Y 390.033,Z 144.902,A -85,B 0,C 180,E1 -11552.722,E2 -11552.722} C_VEL
LIN {X 0,Y 390.047,Z 144.898,A -85,B 0,C 180,E1 -11555.826,E2 -11555.826} C_VEL
LIN {X 0,Y 390.059,Z 144.895,A -85,B 0,C 180,E1 -11559.219,E2 -11559.219} C_VEL
LIN {X 0,Y 390.035,Z 144.903,A -85,B 0,C 180,E1 -11562.375,E2 -11562.375} C_VEL
LIN {X 0,Y 390.037,Z 144.897,A -85,B 0,C 180,E1 -11565.355,E2 -11565.355} C_VEL
LIN {X 0,Y 390.025,Z 144.905,A -85,B 0,C 180,E1 -11568.188,E2 -11568.188} C_VEL
LIN {X 0,Y 390.086,Z 144.891,A -85,B 0,C 180,E1 -11570.909,E2 -11570.909} C_VEL
LIN {X 0,Y 390.08,Z 144.892,A -85,B 0,C 180,E1 -11574.794,E2 -11574.794} C_VEL
LIN {X 0,Y 390.028,Z 144.903,A -85,B 0,C 180,E1 -11577.877,E2 -11577.877} C_VEL
LIN {X 0,Y 390.143,Z 145.009,A -85,B 0,C 180,E1 -11581.297,E2 -11581.297} C_VEL
LIN {X 0,Y 392.648,Z 157.363,A -85,B 0,C 180,E1 -11584.047,E2 -11584.047} C_VEL
LIN {X 0,Y 393.23,Z 162.623,A -85,B 0,C 180,E1 -11585.167,E2 -11585.167} C_VEL
LIN {X 0,Y 392.022,Z 178.92,A -85,B 0,C 180,E1 -11588.439,E2 -11588.439} C_VEL
LIN {X 0,Y 391.557,Z 186.746,A -85,B 0,C 180,E1 -11589.976,E2 -11589.976} C_VEL
LIN {X 0,Y 395.891,Z 218.199,A -85,B 0,C 180,E1 -11590.765,E2 -11590.765} C_VEL
LIN {X 0,Y 394.956,Z 295.745,A -85,B 0,C 180,E1 -11592.193,E2 -11592.193} C_VEL
LIN {X 0,Y 394.281,Z 309.669,A -85,B 0,C 180,E1 -11592.663,E2 -11592.663} C_VEL
LIN {X 0,Y 393.637,Z 321.606,A -85,B 0,C 180,E1 -11593.269,E2 -11593.269} C_VEL
LIN {X 0,Y 392.872,Z 332.883,A -85,B 0,C 180,E1 -11594.037,E2 -11594.037} C_VEL
LIN {X 0,Y 392.019,Z 344.573,A -85,B 0,C 180,E1 -11595.067,E2 -11595.067} C_VEL
LIN {X 0,Y 391.24,Z 355.383,A -85,B 0,C 180,E1 -11596.267,E2 -11596.267} C_VEL
LIN {X 0,Y 390.468,Z 364.554,A -85,B 0,C 180,E1 -11597.528,E2 -11597.528} C_VEL
LIN {X 0,Y 389.729,Z 373.681,A -85,B 0,C 180,E1 -11599.086,E2 -11599.086} C_VEL
LIN {X 0,Y 389.255,Z 381.039,A -85,B 0,C 180,E1 -11600.649,E2 -11600.649} C_VEL
LIN {X 0,Y 388.963,Z 386.934,A -85,B 0,C 180,E1 -11602.213,E2 -11602.213} C_VEL
LIN {X 0,Y 388.774,Z 391.777,A -85,B 0,C 180,E1 -11603.856,E2 -11603.856} C_VEL
LIN {X 0,Y 388.73,Z 395.091,A -85,B 0,C 180,E1 -11605.334,E2 -11605.334} C_VEL
LIN {X 0,Y 388.712,Z 397.594,A -85,B 0,C 180,E1 -11606.892,E2 -11606.892} C_VEL
LIN {X 0,Y 388.795,Z 398.748,A -85,B 0,C 180,E1 -11607.929,E2 -11607.929} C_VEL
LIN {X 0,Y 388.764,Z 399.462,A -85,B 0,C 180,E1 -11608.965,E2 -11608.965} C_VEL
LIN {X 0,Y 388.752,Z 399.788,A -85,B 0,C 180,E1 -11610.001,E2 -11610.001} C_VEL
LIN {X 0,Y 388.763,Z 399.728,A -85,B 0,C 180,E1 -11611.037,E2 -11611.037} C_VEL
LIN {X 0,Y 388.756,Z 399.265,A -85,B 0,C 180,E1 -11612.073,E2 -11612.073} C_VEL
LIN {X 0,Y 388.702,Z 397.076,A -85,B 0,C 180,E1 -11614.148,E2 -11614.148} C_VEL
LIN {X 0,Y 388.729,Z 393.57,A -85,B 0,C 180,E1 -11616.082,E2 -11616.082} C_VEL
LIN {X 0,Y 388.988,Z 389.141,A -85,B 0,C 180,E1 -11617.789,E2 -11617.789} C_VEL
LIN {X 0,Y 389.41,Z 382.872,A -85,B 0,C 180,E1 -11619.611,E2 -11619.611} C_VEL
LIN {X 0,Y 389.969,Z 376.066,A -85,B 0,C 180,E1 -11621.172,E2 -11621.172} C_VEL
LIN {X 0,Y 390.901,Z 367.629,A -85,B 0,C 180,E1 -11622.724,E2 -11622.724} C_VEL
LIN {X 0,Y 391.745,Z 357.701,A -85,B 0,C 180,E1 -11624.186,E2 -11624.186} C_VEL
LIN {X 0,Y 392.775,Z 347.119,A -85,B 0,C 180,E1 -11625.437,E2 -11625.437} C_VEL
LIN {X 0,Y 393.849,Z 336.204,A -85,B 0,C 180,E1 -11626.457,E2 -11626.457} C_VEL
LIN {X 0,Y 394.867,Z 323.984,A -85,B 0,C 180,E1 -11627.346,E2 -11627.346} C_VEL
LIN {X 0,Y 395.746,Z 312.47,A -85,B 0,C 180,E1 -11627.973,E2 -11627.973} C_VEL
LIN {X 0,Y 396.435,Z 300.421,A -85,B 0,C 180,E1 -11628.442,E2 -11628.442} C_VEL
LIN {X 0,Y 396.817,Z 285.598,A -85,B 0,C 180,E1 -11628.787,E2 -11628.787} C_VEL
LIN {X 0,Y 397.693,Z 218.213,A -85,B 0,C 180,E1 -11630.017,E2 -11630.017} C_VEL
LIN {X 0,Y 394.291,Z 196.778,A -85,B 0,C 180,E1 -11630.625,E2 -11630.625} C_VEL
LIN {X 0,Y 392.348,Z 186.329,A -85,B 0,C 180,E1 -11630.945,E2 -11630.945} C_VEL
LIN {X 0,Y 393.824,Z 168.994,A -85,B 0,C 180,E1 -11634.477,E2 -11634.477} C_VEL
LIN {X 0,Y 394.041,Z 163.496,A -85,B 0,C 180,E1 -11635.628,E2 -11635.628} C_VEL
LIN {X 0,Y 391.577,Z 151.333,A -85,B 0,C 180,E1 -11638.424,E2 -11638.424} C_VEL
LIN {X 0,Y 390.068,Z 144.904,A -85,B 0,C 180,E1 -11639.974,E2 -11639.974} C_VEL
LIN {X 0,Y 390.071,Z 144.9,A -85,B 0,C 180,E1 -11643.955,E2 -11643.955} C_VEL
LIN {X 0,Y 390.059,Z 144.894,A -85,B 0,C 180,E1 -11646.484,E2 -11646.484} C_VEL
LIN {X 0,Y 390.063,Z 144.893,A -85,B 0,C 180,E1 -11649.217,E2 -11649.217} C_VEL
LIN {X 0,Y 390.041,Z 144.896,A -85,B 0,C 180,E1 -11652.374,E2 -11652.374} C_VEL
LIN {X 0,Y 390.046,Z 144.901,A -85,B 0,C 180,E1 -11655.354,E2 -11655.354} C_VEL
LIN {X 0,Y 390.022,Z 144.901,A -85,B 0,C 180,E1 -11658.185,E2 -11658.185} C_VEL
LIN {X 0,Y 390.059,Z 144.899,A -85,B 0,C 180,E1 -11660.904,E2 -11660.904} C_VEL
LIN {X 0,Y 390.071,Z 144.898,A -85,B 0,C 180,E1 -11664.792,E2 -11664.792} C_VEL
LIN {X 0,Y 390.024,Z 144.902,A -85,B 0,C 180,E1 -11668.496,E2 -11668.496} C_VEL
LIN {X 0,Y 390.029,Z 144.898,A -85,B 0,C 180,E1 -11672.063,E2 -11672.063} C_VEL
LIN {X 0,Y 390.043,Z 144.897,A -85,B 0,C 180,E1 -11675.517,E2 -11675.517} C_VEL
LIN {X 0,Y 390.053,Z 144.895,A -85,B 0,C 180,E1 -11678.878,E2 -11678.878} C_VEL
LIN {X 0,Y 390.068,Z 144.893,A -85,B 0,C 180,E1 -11682.164,E2 -11682.164} C_VEL
LIN {X 0,Y 390.069,Z 144.886,A -85,B 0,C 180,E1 -11685.39,E2 -11685.39} C_VEL
LIN {X 0,Y 390.166,Z 144.88,A -85,B 0,C 180,E1 -11687.517,E2 -11687.517} C_VEL
LIN {X 0,Y 390.184,Z 144.873,A -85,B 0,C 180,E1 -11690.671,E2 -11690.671} C_VEL
LIN {X 0,Y 390.274,Z 144.87,A -85,B 0,C 180,E1 -11693.797,E2 -11693.797} C_VEL
LIN {X 0,Y 390.403,Z 144.848,A -85,B 0,C 180,E1 -11697.937,E2 -11697.937} C_VEL
LIN {X 0,Y 390.404,Z 144.847,A -85,B 0,C 180,E1 -11702.063,E2 -11702.063} C_VEL
LIN {X 0,Y 390.262,Z 144.869,A -85,B 0,C 180,E1 -11706.453,E2 -11706.453} C_VEL
LIN {X 0,Y 390.193,Z 144.872,A -85,B 0,C 180,E1 -11709.329,E2 -11709.329} C_VEL
LIN {X 0,Y 390.171,Z 144.88,A -85,B 0,C 180,E1 -11712.483,E2 -11712.483} C_VEL
LIN {X 0,Y 390.139,Z 144.888,A -85,B 0,C 180,E1 -11715.677,E2 -11715.677} C_VEL
LIN {X 0,Y 390.103,Z 144.889,A -85,B 0,C 180,E1 -11718.922,E2 -11718.922} C_VEL
LIN {X 0,Y 390.038,Z 144.898,A -85,B 0,C 180,E1 -11722.234,E2 -11722.234} C_VEL
LIN {X 0,Y 390.069,Z 144.894,A -85,B 0,C 180,E1 -11725.727,E2 -11725.727} C_VEL
LIN {X 0,Y 390.046,Z 144.897,A -85,B 0,C 180,E1 -11729.111,E2 -11729.111} C_VEL
LIN {X 0,Y 390.045,Z 144.897,A -85,B 0,C 180,E1 -11732.722,E2 -11732.722} C_VEL
LIN {X 0,Y 390.058,Z 144.894,A -85,B 0,C 180,E1 -11735.825,E2 -11735.825} C_VEL
LIN {X 0,Y 390.069,Z 144.891,A -85,B 0,C 180,E1 -11739.218,E2 -11739.218} C_VEL
LIN {X 0,Y 390.045,Z 144.89,A -85,B 0,C 180,E1 -11742.374,E2 -11742.374} C_VEL
LIN {X 0,Y 390.047,Z 144.895,A -85,B 0,C 180,E1 -11745.354,E2 -11745.354} C_VEL
LIN {X 0,Y 390.028,Z 144.903,A -85,B 0,C 180,E1 -11748.186,E2 -11748.186} C_VEL
LIN {X 0,Y 390.086,Z 144.893,A -85,B 0,C 180,E1 -11750.907,E2 -11750.907} C_VEL
LIN {X 0,Y 390.089,Z 144.893,A -85,B 0,C 180,E1 -11754.793,E2 -11754.793} C_VEL
LIN {X 0,Y 390.028,Z 144.899,A -85,B 0,C 180,E1 -11758.495,E2 -11758.495} C_VEL
LIN {X 0,Y 390.093,Z 144.895,A -85,B 0,C 180,E1 -11761.724,E2 -11761.724} C_VEL
LIN {X 0,Y 392.067,Z 154.091,A -85,B 0,C 180,E1 -11764.089,E2 -11764.089} C_VEL
LIN {X 0,Y 395.674,Z 164.126,A -85,B 0,C 180,E1 -11764.505,E2 -11764.505} C_VEL
LIN {X 0,Y 398.387,Z 175.912,A -85,B 0,C 180,E1 -11764.894,E2 -11764.894} C_VEL
LIN {X 0,Y 397.074,Z 260.96,A -85,B 0,C 180,E1 -11766.462,E2 -11766.462} C_VEL
LIN {X 0,Y 396.51,Z 274.326,A -85,B 0,C 180,E1 -11766.911,E2 -11766.911} C_VEL
LIN {X 0,Y 395.865,Z 287.019,A -85,B 0,C 180,E1 -11767.554,E2 -11767.554} C_VEL
LIN {X 0,Y 395.153,Z 298.44,A -85,B 0,C 180,E1 -11768.342,E2 -11768.342} C_VEL
LIN {X 0,Y 394.142,Z 310.1,A -85,B 0,C 180,E1 -11769.38,E2 -11769.38} C_VEL
LIN {X 0,Y 393.171,Z 320.56,A -85,B 0,C 180,E1 -11770.553,E2 -11770.553} C_VEL
LIN {X 0,Y 392.301,Z 329.97,A -85,B 0,C 180,E1 -11771.87,E2 -11771.87} C_VEL
LIN {X 0,Y 391.414,Z 338.273,A -85,B 0,C 180,E1 -11773.304,E2 -11773.304} C_VEL
LIN {X 0,Y 390.602,Z 345.638,A -85,B 0,C 180,E1 -11774.876,E2 -11774.876} C_VEL
LIN {X 0,Y 389.992,Z 351.52,A -85,B 0,C 180,E1 -11776.451,E2 -11776.451} C_VEL
LIN {X 0,Y 389.515,Z 356.141,A -85,B 0,C 180,E1 -11778.024,E2 -11778.024} C_VEL
LIN {X 0,Y 389.12,Z 359.647,A -85,B 0,C 180,E1 -11779.594,E2 -11779.594} C_VEL
LIN {X 0,Y 388.989,Z 361.417,A -85,B 0,C 180,E1 -11780.641,E2 -11780.641} C_VEL
LIN {X 0,Y 388.901,Z 363.68,A -85,B 0,C 180,E1 -11782.732,E2 -11782.732} C_VEL
LIN {X 0,Y 388.878,Z 364.231,A -85,B 0,C 180,E1 -11783.774,E2 -11783.774} C_VEL
LIN {X 0,Y 388.824,Z 364.362,A -85,B 0,C 180,E1 -11784.814,E2 -11784.814} C_VEL
LIN {X 0,Y 388.805,Z 363.446,A -85,B 0,C 180,E1 -11786.891,E2 -11786.891} C_VEL
LIN {X 0,Y 388.864,Z 362.415,A -85,B 0,C 180,E1 -11787.928,E2 -11787.928} C_VEL
LIN {X 0,Y 388.84,Z 360.959,A -85,B 0,C 180,E1 -11788.963,E2 -11788.963} C_VEL
LIN {X 0,Y 389.057,Z 357.985,A -85,B 0,C 180,E1 -11790.517,E2 -11790.517} C_VEL
LIN {X 0,Y 389.276,Z 353.982,A -85,B 0,C 180,E1 -11792.068,E2 -11792.068} C_VEL
LIN {X 0,Y 389.685,Z 348.824,A -85,B 0,C 180,E1 -11793.618,E2 -11793.618} C_VEL
LIN {X 0,Y 390.193,Z 342.354,A -85,B 0,C 180,E1 -11795.166,E2 -11795.166} C_VEL
LIN {X 0,Y 390.956,Z 334.306,A -85,B 0,C 180,E1 -11796.709,E2 -11796.709} C_VEL
LIN {X 0,Y 391.703,Z 325.569,A -85,B 0,C 180,E1 -11798.066,E2 -11798.066} C_VEL
LIN {X 0,Y 391.255,Z 322.747,A -85,B 0,C 180,E1 -11798.474,E2 -11798.474} C_VEL
LIN {X 0,Y 386.421,Z 313.714,A -85,B 0,C 180,E1 -11799.772,E2 -11799.772} C_VEL
LIN {X 0,Y 386.021,Z 310.553,A -85,B 0,C 180,E1 -11800.128,E2 -11800.128} C_VEL
LIN {X 0,Y 386.773,Z 299.756,A -85,B 0,C 180,E1 -11801.118,E2 -11801.118} C_VEL
LIN {X 0,Y 387.45,Z 287.848,A -85,B 0,C 180,E1 -11801.973,E2 -11801.973} C_VEL
LIN {X 0,Y 387.995,Z 274.835,A -85,B 0,C 180,E1 -11802.653,E2 -11802.653} C_VEL
LIN {X 0,Y 388.395,Z 261.941,A -85,B 0,C 180,E1 -11803.105,E2 -11803.105} C_VEL
LIN {X 0,Y 389.634,Z 180.508,A -85,B 0,C 180,E1 -11804.626,E2 -11804.626} C_VEL
LIN {X 0,Y 389.398,Z 174.599,A -85,B 0,C 180,E1 -11804.749,E2 -11804.749} C_VEL
LIN {X 0,Y 385.565,Z 156.382,A -85,B 0,C 180,E1 -11805.287,E2 -11805.287} C_VEL
LIN {X 0,Y 384.687,Z 153.796,A -85,B 0,C 180,E1 -11805.41,E2 -11805.41} C_VEL
LIN {X 0,Y 383.096,Z 145.766,A -85,B 0,C 180,E1 -11807.503,E2 -11807.503} C_VEL
LIN {X 0,Y 383.029,Z 145.773,A -85,B 0,C 180,E1 -11810.646,E2 -11810.646} C_VEL
LIN {X 0,Y 383.022,Z 145.773,A -85,B 0,C 180,E1 -11813.807,E2 -11813.807} C_VEL
LIN {X 0,Y 383.078,Z 145.769,A -85,B 0,C 180,E1 -11816.122,E2 -11816.122} C_VEL
LIN {X 0,Y 383.039,Z 145.772,A -85,B 0,C 180,E1 -11818.491,E2 -11818.491} C_VEL
LIN {X 0,Y 383.007,Z 145.779,A -85,B 0,C 180,E1 -11822.148,E2 -11822.148} C_VEL
LIN {X 0,Y 383.015,Z 145.773,A -85,B 0,C 180,E1 -11824.666,E2 -11824.666} C_VEL
LIN {X 0,Y 382.996,Z 145.78,A -85,B 0,C 180,E1 -11827.902,E2 -11827.902} C_VEL
LIN {X 0,Y 382.979,Z 145.777,A -85,B 0,C 180,E1 -11831.346,E2 -11831.346} C_VEL
LIN {X 0,Y 382.99,Z 145.778,A -85,B 0,C 180,E1 -11834.302,E2 -11834.302} C_VEL
LIN {X 0,Y 383.004,Z 145.774,A -85,B 0,C 180,E1 -11837.239,E2 -11837.239} C_VEL
LIN {X 0,Y 383.006,Z 145.774,A -85,B 0,C 180,E1 -11840.413,E2 -11840.413} C_VEL
LIN {X 0,Y 383.017,Z 145.775,A -85,B 0,C 180,E1 -11844.043,E2 -11844.043} C_VEL
LIN {X 0,Y 382.978,Z 145.782,A -85,B 0,C 180,E1 -11847.577,E2 -11847.577} C_VEL
LIN {X 0,Y 382.983,Z 145.777,A -85,B 0,C 180,E1 -11850.299,E2 -11850.299} C_VEL
LIN {X 0,Y 383.04,Z 145.772,A -85,B 0,C 180,E1 -11853.873,E2 -11853.873} C_VEL
LIN {X 0,Y 382.981,Z 145.782,A -85,B 0,C 180,E1 -11857.333,E2 -11857.333} C_VEL
LIN {X 0,Y 383.047,Z 145.769,A -85,B 0,C 180,E1 -11860.715,E2 -11860.715} C_VEL
LIN {X 0,Y 383.065,Z 145.767,A -85,B 0,C 180,E1 -11864.026,E2 -11864.026} C_VEL
LIN {X 0,Y 383.125,Z 145.763,A -85,B 0,C 180,E1 -11867.283,E2 -11867.283} C_VEL
LIN {X 0,Y 383.131,Z 145.758,A -85,B 0,C 180,E1 -11870.497,E2 -11870.497} C_VEL
LIN {X 0,Y 383.221,Z 145.748,A -85,B 0,C 180,E1 -11873.682,E2 -11873.682} C_VEL
LIN {X 0,Y 383.36,Z 145.73,A -85,B 0,C 180,E1 -11877.899,E2 -11877.899} C_VEL
LIN {X 0,Y 383.36,Z 145.729,A -85,B 0,C 180,E1 -11882.101,E2 -11882.101} C_VEL
LIN {X 0,Y 383.228,Z 145.747,A -85,B 0,C 180,E1 -11886.317,E2 -11886.317} C_VEL
LIN {X 0,Y 383.131,Z 145.759,A -85,B 0,C 180,E1 -11889.503,E2 -11889.503} C_VEL
LIN {X 0,Y 383.114,Z 145.76,A -85,B 0,C 180,E1 -11893.536,E2 -11893.536} C_VEL
LIN {X 0,Y 383.083,Z 145.767,A -85,B 0,C 180,E1 -11897.07,E2 -11897.07} C_VEL
LIN {X 0,Y 383.018,Z 145.777,A -85,B 0,C 180,E1 -11900.647,E2 -11900.647} C_VEL
LIN {X 0,Y 383.007,Z 145.774,A -85,B 0,C 180,E1 -11903.809,E2 -11903.809} C_VEL
LIN {X 0,Y 383.045,Z 145.769,A -85,B 0,C 180,E1 -11907.303,E2 -11907.303} C_VEL
LIN {X 0,Y 382.973,Z 145.779,A -85,B 0,C 180,E1 -11910.919,E2 -11910.919} C_VEL
LIN {X 0,Y 383.009,Z 145.776,A -85,B 0,C 180,E1 -11914.669,E2 -11914.669} C_VEL
LIN {X 0,Y 382.99,Z 145.777,A -85,B 0,C 180,E1 -11917.904,E2 -11917.904} C_VEL
LIN {X 0,Y 382.976,Z 145.777,A -85,B 0,C 180,E1 -11921.349,E2 -11921.349} C_VEL
LIN {X 0,Y 382.989,Z 145.781,A -85,B 0,C 180,E1 -11924.304,E2 -11924.304} C_VEL
LIN {X 0,Y 383.004,Z 145.773,A -85,B 0,C 180,E1 -11927.241,E2 -11927.241} C_VEL
LIN {X 0,Y 383.01,Z 145.776,A -85,B 0,C 180,E1 -11930.415,E2 -11930.415} C_VEL
LIN {X 0,Y 383.02,Z 145.777,A -85,B 0,C 180,E1 -11934.046,E2 -11934.046} C_VEL
LIN {X 0,Y 382.983,Z 145.778,A -85,B 0,C 180,E1 -11937.579,E2 -11937.579} C_VEL
LIN {X 0,Y 383.082,Z 145.875,A -85,B 0,C 180,E1 -11941.025,E2 -11941.025} C_VEL
LIN {X 0,Y 385.507,Z 157.781,A -85,B 0,C 180,E1 -11943.733,E2 -11943.733} C_VEL
LIN {X 0,Y 386.287,Z 163.471,A -85,B 0,C 180,E1 -11944.977,E2 -11944.977} C_VEL
LIN {X 0,Y 385.047,Z 179.763,A -85,B 0,C 180,E1 -11948.31,E2 -11948.31} C_VEL
LIN {X 0,Y 384.601,Z 186.295,A -85,B 0,C 180,E1 -11949.634,E2 -11949.634} C_VEL
LIN {X 0,Y 389.103,Z 218.89,A -85,B 0,C 180,E1 -11950.47,E2 -11950.47} C_VEL
LIN {X 0,Y 388.143,Z 295.382,A -85,B 0,C 180,E1 -11951.903,E2 -11951.903} C_VEL
LIN {X 0,Y 387.462,Z 309.322,A -85,B 0,C 180,E1 -11952.382,E2 -11952.382} C_VEL
LIN {X 0,Y 386.735,Z 321.808,A -85,B 0,C 180,E1 -11953.03,E2 -11953.03} C_VEL
LIN {X 0,Y 385.883,Z 333.742,A -85,B 0,C 180,E1 -11953.876,E2 -11953.876} C_VEL
LIN {X 0,Y 385.017,Z 345.218,A -85,B 0,C 180,E1 -11954.924,E2 -11954.924} C_VEL
LIN {X 0,Y 384.252,Z 355.286,A -85,B 0,C 180,E1 -11956.075,E2 -11956.075} C_VEL
LIN {X 0,Y 383.464,Z 364.015,A -85,B 0,C 180,E1 -11957.296,E2 -11957.296} C_VEL
LIN {X 0,Y 382.697,Z 373.181,A -85,B 0,C 180,E1 -11958.883,E2 -11958.883} C_VEL
LIN {X 0,Y 382.192,Z 380.571,A -85,B 0,C 180,E1 -11960.475,E2 -11960.475} C_VEL
LIN {X 0,Y 381.882,Z 386.494,A -85,B 0,C 180,E1 -11962.067,E2 -11962.067} C_VEL
LIN {X 0,Y 381.671,Z 391.761,A -85,B 0,C 180,E1 -11963.905,E2 -11963.905} C_VEL
LIN {X 0,Y 381.647,Z 395.634,A -85,B 0,C 180,E1 -11965.777,E2 -11965.777} C_VEL
LIN {X 0,Y 381.617,Z 397.224,A -85,B 0,C 180,E1 -11966.834,E2 -11966.834} C_VEL
LIN {X 0,Y 381.695,Z 398.397,A -85,B 0,C 180,E1 -11967.891,E2 -11967.891} C_VEL
LIN {X 0,Y 381.695,Z 399.124,A -85,B 0,C 180,E1 -11968.946,E2 -11968.946} C_VEL
LIN {X 0,Y 381.694,Z 399.41,A -85,B 0,C 180,E1 -11971.056,E2 -11971.056} C_VEL
LIN {X 0,Y 381.654,Z 398.963,A -85,B 0,C 180,E1 -11972.112,E2 -11972.112} C_VEL
LIN {X 0,Y 381.625,Z 396.797,A -85,B 0,C 180,E1 -11974.225,E2 -11974.225} C_VEL
LIN {X 0,Y 381.627,Z 393.642,A -85,B 0,C 180,E1 -11976.033,E2 -11976.033} C_VEL
LIN {X 0,Y 381.914,Z 388.915,A -85,B 0,C 180,E1 -11977.934,E2 -11977.934} C_VEL
LIN {X 0,Y 382.362,Z 382.673,A -85,B 0,C 180,E1 -11979.79,E2 -11979.79} C_VEL
LIN {X 0,Y 382.957,Z 375.897,A -85,B 0,C 180,E1 -11981.379,E2 -11981.379} C_VEL
LIN {X 0,Y 383.956,Z 367.507,A -85,B 0,C 180,E1 -11982.958,E2 -11982.958} C_VEL
LIN {X 0,Y 384.849,Z 357.627,A -85,B 0,C 180,E1 -11984.446,E2 -11984.446} C_VEL
LIN {X 0,Y 385.938,Z 347.098,A -85,B 0,C 180,E1 -11985.717,E2 -11985.717} C_VEL
LIN {X 0,Y 387.051,Z 336.288,A -85,B 0,C 180,E1 -11986.754,E2 -11986.754} C_VEL
LIN {X 0,Y 388.107,Z 324.174,A -85,B 0,C 180,E1 -11987.658,E2 -11987.658} C_VEL
LIN {X 0,Y 389.006,Z 312.819,A -85,B 0,C 180,E1 -11988.296,E2 -11988.296} C_VEL
LIN {X 0,Y 389.77,Z 300.135,A -85,B 0,C 180,E1 -11988.803,E2 -11988.803} C_VEL
LIN {X 0,Y 390.186,Z 285.527,A -85,B 0,C 180,E1 -11989.149,E2 -11989.149} C_VEL
LIN {X 0,Y 391.04,Z 218.719,A -85,B 0,C 180,E1 -11990.393,E2 -11990.393} C_VEL
LIN {X 0,Y 387.763,Z 197.976,A -85,B 0,C 180,E1 -11990.996,E2 -11990.996} C_VEL
LIN {X 0,Y 385.512,Z 185.939,A -85,B 0,C 180,E1 -11991.384,E2 -11991.384} C_VEL
LIN {X 0,Y 387.039,Z 168.807,A -85,B 0,C 180,E1 -11994.944,E2 -11994.944} C_VEL
LIN {X 0,Y 387.26,Z 166.015,A -85,B 0,C 180,E1 -11995.532,E2 -11995.532} C_VEL
LIN {X 0,Y 385.501,Z 156.647,A -85,B 0,C 180,E1 -11997.703,E2 -11997.703} C_VEL
LIN {X 0,Y 383.003,Z 145.784,A -85,B 0,C 180,E1 -12000.35,E2 -12000.35} C_VEL
LIN {X 0,Y 383.006,Z 145.779,A -85,B 0,C 180,E1 -12003.401,E2 -12003.401} C_VEL
LIN {X 0,Y 383.034,Z 145.771,A -85,B 0,C 180,E1 -12006.165,E2 -12006.165} C_VEL
LIN {X 0,Y 382.996,Z 145.777,A -85,B 0,C 180,E1 -12009.961,E2 -12009.961} C_VEL
LIN {X 0,Y 383.008,Z 145.772,A -85,B 0,C 180,E1 -12012.779,E2 -12012.779} C_VEL
LIN {X 0,Y 382.998,Z 145.778,A -85,B 0,C 180,E1 -12015.789,E2 -12015.789} C_VEL
LIN {X 0,Y 382.965,Z 145.781,A -85,B 0,C 180,E1 -12018.8,E2 -12018.8} C_VEL
LIN {X 0,Y 382.995,Z 145.776,A -85,B 0,C 180,E1 -12022.098,E2 -12022.098} C_VEL
LIN {X 0,Y 383.013,Z 145.778,A -85,B 0,C 180,E1 -12025.331,E2 -12025.331} C_VEL
LIN {X 0,Y 382.983,Z 145.78,A -85,B 0,C 180,E1 -12029.081,E2 -12029.081} C_VEL
LIN {X 0,Y 382.986,Z 145.78,A -85,B 0,C 180,E1 -12032.693,E2 -12032.693} C_VEL
LIN {X 0,Y 383.011,Z 145.774,A -85,B 0,C 180,E1 -12036.191,E2 -12036.191} C_VEL
LIN {X 0,Y 383.041,Z 145.765,A -85,B 0,C 180,E1 -12039.598,E2 -12039.598} C_VEL
LIN {X 0,Y 383.07,Z 145.767,A -85,B 0,C 180,E1 -12042.93,E2 -12042.93} C_VEL
LIN {X 0,Y 383.128,Z 145.756,A -85,B 0,C 180,E1 -12047.284,E2 -12047.284} C_VEL
LIN {X 0,Y 383.135,Z 145.753,A -85,B 0,C 180,E1 -12050.498,E2 -12050.498} C_VEL
LIN {X 0,Y 383.232,Z 145.746,A -85,B 0,C 180,E1 -12053.683,E2 -12053.683} C_VEL
LIN {X 0,Y 383.367,Z 145.724,A -85,B 0,C 180,E1 -12057.899,E2 -12057.899} C_VEL
LIN {X 0,Y 383.369,Z 145.723,A -85,B 0,C 180,E1 -12062.101,E2 -12062.101} C_VEL
LIN {X 0,Y 383.227,Z 145.745,A -85,B 0,C 180,E1 -12066.44,E2 -12066.44} C_VEL
LIN {X 0,Y 383.143,Z 145.752,A -85,B 0,C 180,E1 -12069.502,E2 -12069.502} C_VEL
LIN {X 0,Y 383.127,Z 145.754,A -85,B 0,C 180,E1 -12073.536,E2 -12073.536} C_VEL
LIN {X 0,Y 383.095,Z 145.766,A -85,B 0,C 180,E1 -12077.069,E2 -12077.069} C_VEL
LIN {X 0,Y 383.03,Z 145.767,A -85,B 0,C 180,E1 -12080.647,E2 -12080.647} C_VEL
LIN {X 0,Y 383.016,Z 145.767,A -85,B 0,C 180,E1 -12083.809,E2 -12083.809} C_VEL
LIN {X 0,Y 383.021,Z 145.772,A -85,B 0,C 180,E1 -12087.305,E2 -12087.305} C_VEL
LIN {X 0,Y 382.984,Z 145.781,A -85,B 0,C 180,E1 -12090.919,E2 -12090.919} C_VEL
LIN {X 0,Y 383.02,Z 145.777,A -85,B 0,C 180,E1 -12094.668,E2 -12094.668} C_VEL
LIN {X 0,Y 383,Z 145.774,A -85,B 0,C 180,E1 -12097.903,E2 -12097.903} C_VEL
LIN {X 0,Y 382.986,Z 145.762,A -85,B 0,C 180,E1 -12101.347,E2 -12101.347} C_VEL
LIN {X 0,Y 382.999,Z 145.779,A -85,B 0,C 180,E1 -12104.303,E2 -12104.303} C_VEL
LIN {X 0,Y 383.014,Z 145.773,A -85,B 0,C 180,E1 -12107.24,E2 -12107.24} C_VEL
LIN {X 0,Y 383.013,Z 145.777,A -85,B 0,C 180,E1 -12110.414,E2 -12110.414} C_VEL
LIN {X 0,Y 383.029,Z 145.775,A -85,B 0,C 180,E1 -12114.044,E2 -12114.044} C_VEL
LIN {X 0,Y 382.991,Z 145.78,A -85,B 0,C 180,E1 -12117.578,E2 -12117.578} C_VEL
LIN {X 0,Y 383.062,Z 145.883,A -85,B 0,C 180,E1 -12121.396,E2 -12121.396} C_VEL
LIN {X 0,Y 384.887,Z 154.179,A -85,B 0,C 180,E1 -12123.623,E2 -12123.623} C_VEL
LIN {X 0,Y 389.187,Z 165.756,A -85,B 0,C 180,E1 -12124.137,E2 -12124.137} C_VEL
LIN {X 0,Y 391.814,Z 177.069,A -85,B 0,C 180,E1 -12124.521,E2 -12124.521} C_VEL
LIN {X 0,Y 390.446,Z 261.579,A -85,B 0,C 180,E1 -12126.108,E2 -12126.108} C_VEL
LIN {X 0,Y 389.863,Z 274.846,A -85,B 0,C 180,E1 -12126.564,E2 -12126.564} C_VEL
LIN {X 0,Y 389.162,Z 287.789,A -85,B 0,C 180,E1 -12127.235,E2 -12127.235} C_VEL
LIN {X 0,Y 388.378,Z 299.661,A -85,B 0,C 180,E1 -12128.085,E2 -12128.085} C_VEL
LIN {X 0,Y 387.31,Z 311.154,A -85,B 0,C 180,E1 -12129.138,E2 -12129.138} C_VEL
LIN {X 0,Y 386.307,Z 321.479,A -85,B 0,C 180,E1 -12130.331,E2 -12130.331} C_VEL
LIN {X 0,Y 385.418,Z 330.555,A -85,B 0,C 180,E1 -12131.639,E2 -12131.639} C_VEL
LIN {X 0,Y 384.547,Z 338.299,A -85,B 0,C 180,E1 -12132.997,E2 -12132.997} C_VEL
LIN {X 0,Y 383.676,Z 345.716,A -85,B 0,C 180,E1 -12134.596,E2 -12134.596} C_VEL
LIN {X 0,Y 383.015,Z 351.646,A -85,B 0,C 180,E1 -12136.199,E2 -12136.199} C_VEL
LIN {X 0,Y 382.51,Z 356.308,A -85,B 0,C 180,E1 -12137.801,E2 -12137.801} C_VEL
LIN {X 0,Y 382.08,Z 359.854,A -85,B 0,C 180,E1 -12139.4,E2 -12139.4} C_VEL
LIN {X 0,Y 381.926,Z 361.662,A -85,B 0,C 180,E1 -12140.466,E2 -12140.466} C_VEL
LIN {X 0,Y 381.818,Z 363.96,A -85,B 0,C 180,E1 -12142.596,E2 -12142.596} C_VEL
LIN {X 0,Y 381.812,Z 364.551,A -85,B 0,C 180,E1 -12143.711,E2 -12143.711} C_VEL
LIN {X 0,Y 381.745,Z 364.695,A -85,B 0,C 180,E1 -12144.718,E2 -12144.718} C_VEL
LIN {X 0,Y 381.707,Z 363.814,A -85,B 0,C 180,E1 -12146.833,E2 -12146.833} C_VEL
LIN {X 0,Y 381.777,Z 362.801,A -85,B 0,C 180,E1 -12147.889,E2 -12147.889} C_VEL
LIN {X 0,Y 381.768,Z 361.38,A -85,B 0,C 180,E1 -12148.944,E2 -12148.944} C_VEL
LIN {X 0,Y 381.992,Z 358.44,A -85,B 0,C 180,E1 -12150.526,E2 -12150.526} C_VEL
LIN {X 0,Y 382.197,Z 354.477,A -85,B 0,C 180,E1 -12152.107,E2 -12152.107} C_VEL
LIN {X 0,Y 382.641,Z 349.367,A -85,B 0,C 180,E1 -12153.685,E2 -12153.685} C_VEL
LIN {X 0,Y 383.159,Z 342.946,A -85,B 0,C 180,E1 -12155.261,E2 -12155.261} C_VEL
LIN {X 0,Y 383.946,Z 334.953,A -85,B 0,C 180,E1 -12156.832,E2 -12156.832} C_VEL
LIN {X 0,Y 384.729,Z 326.174,A -85,B 0,C 180,E1 -12158.23,E2 -12158.23} C_VEL
LIN {X 0,Y 385.559,Z 316.85,A -85,B 0,C 180,E1 -12159.441,E2 -12159.441} C_VEL
LIN {X 0,Y 386.021,Z 310.553,A -85,B 0,C 180,E1 -12160.128,E2 -12160.128} C_VEL
LIN {X 0,Y 385.762,Z 305.71,A -85,B 0,C 180,E1 -12160.627,E2 -12160.627} C_VEL
LIN {X 0,Y 383.509,Z 297.642,A -85,B 0,C 180,E1 -12161.432,E2 -12161.432} C_VEL
LIN {X 0,Y 381.191,Z 289.274,A -85,B 0,C 180,E1 -12162.149,E2 -12162.149} C_VEL
LIN {X 0,Y 380.831,Z 283.888,A -85,B 0,C 180,E1 -12162.503,E2 -12162.503} C_VEL
LIN {X 0,Y 381.369,Z 271.893,A -85,B 0,C 180,E1 -12163.079,E2 -12163.079} C_VEL
LIN {X 0,Y 381.646,Z 259.338,A -85,B 0,C 180,E1 -12163.476,E2 -12163.476} C_VEL
LIN {X 0,Y 382.85,Z 176.621,A -85,B 0,C 180,E1 -12165.032,E2 -12165.032} C_VEL
LIN {X 0,Y 379.147,Z 158.83,A -85,B 0,C 180,E1 -12165.567,E2 -12165.567} C_VEL
LIN {X 0,Y 377.546,Z 154.114,A -85,B 0,C 180,E1 -12165.773,E2 -12165.773} C_VEL
LIN {X 0,Y 376.062,Z 146.641,A -85,B 0,C 180,E1 -12167.736,E2 -12167.736} C_VEL
LIN {X 0,Y 375.978,Z 146.65,A -85,B 0,C 180,E1 -12170.831,E2 -12170.831} C_VEL
LIN {X 0,Y 375.987,Z 146.653,A -85,B 0,C 180,E1 -12174.28,E2 -12174.28} C_VEL
LIN {X 0,Y 376.018,Z 146.646,A -85,B 0,C 180,E1 -12176.651,E2 -12176.651} C_VEL
LIN {X 0,Y 375.968,Z 146.65,A -85,B 0,C 180,E1 -12179.078,E2 -12179.078} C_VEL
LIN {X 0,Y 375.946,Z 146.653,A -85,B 0,C 180,E1 -12182.827,E2 -12182.827} C_VEL
LIN {X 0,Y 375.954,Z 146.652,A -85,B 0,C 180,E1 -12185.414,E2 -12185.414} C_VEL
LIN {X 0,Y 375.971,Z 146.653,A -85,B 0,C 180,E1 -12188.269,E2 -12188.269} C_VEL
LIN {X 0,Y 375.93,Z 146.657,A -85,B 0,C 180,E1 -12191.599,E2 -12191.599} C_VEL
LIN {X 0,Y 375.921,Z 146.657,A -85,B 0,C 180,E1 -12195.267,E2 -12195.267} C_VEL
LIN {X 0,Y 375.927,Z 146.656,A -85,B 0,C 180,E1 -12198.398,E2 -12198.398} C_VEL
LIN {X 0,Y 375.965,Z 146.656,A -85,B 0,C 180,E1 -12201.729,E2 -12201.729} C_VEL
LIN {X 0,Y 375.972,Z 146.652,A -85,B 0,C 180,E1 -12205.332,E2 -12205.332} C_VEL
LIN {X 0,Y 375.949,Z 146.653,A -85,B 0,C 180,E1 -12208.437,E2 -12208.437} C_VEL
LIN {X 0,Y 375.973,Z 146.651,A -85,B 0,C 180,E1 -12212.139,E2 -12212.139} C_VEL
LIN {X 0,Y 375.981,Z 146.648,A -85,B 0,C 180,E1 -12214.537,E2 -12214.537} C_VEL
LIN {X 0,Y 375.946,Z 146.654,A -85,B 0,C 180,E1 -12218.044,E2 -12218.044} C_VEL
LIN {X 0,Y 375.991,Z 146.652,A -85,B 0,C 180,E1 -12221.472,E2 -12221.472} C_VEL
LIN {X 0,Y 376.044,Z 146.642,A -85,B 0,C 180,E1 -12224.832,E2 -12224.832} C_VEL
LIN {X 0,Y 376.036,Z 146.642,A -85,B 0,C 180,E1 -12228.136,E2 -12228.136} C_VEL
LIN {X 0,Y 376.175,Z 146.625,A -85,B 0,C 180,E1 -12231.954,E2 -12231.954} C_VEL
LIN {X 0,Y 376.131,Z 146.631,A -85,B 0,C 180,E1 -12234.639,E2 -12234.639} C_VEL
LIN {X 0,Y 376.325,Z 146.606,A -85,B 0,C 180,E1 -12237.859,E2 -12237.859} C_VEL
LIN {X 0,Y 376.325,Z 146.606,A -85,B 0,C 180,E1 -12242.14,E2 -12242.14} C_VEL
LIN {X 0,Y 376.187,Z 146.624,A -85,B 0,C 180,E1 -12246.436,E2 -12246.436} C_VEL
LIN {X 0,Y 376.101,Z 146.634,A -85,B 0,C 180,E1 -12249.682,E2 -12249.682} C_VEL
LIN {X 0,Y 376.078,Z 146.636,A -85,B 0,C 180,E1 -12253.658,E2 -12253.658} C_VEL
LIN {X 0,Y 376.021,Z 146.644,A -85,B 0,C 180,E1 -12257.4,E2 -12257.4} C_VEL
LIN {X 0,Y 375.968,Z 146.654,A -85,B 0,C 180,E1 -12260.833,E2 -12260.833} C_VEL
LIN {X 0,Y 375.969,Z 146.653,A -85,B 0,C 180,E1 -12264.283,E2 -12264.283} C_VEL
LIN {X 0,Y 375.985,Z 146.648,A -85,B 0,C 180,E1 -12267.86,E2 -12267.86} C_VEL
LIN {X 0,Y 375.948,Z 146.652,A -85,B 0,C 180,E1 -12271.563,E2 -12271.563} C_VEL
LIN {X 0,Y 375.948,Z 146.652,A -85,B 0,C 180,E1 -12275.417,E2 -12275.417} C_VEL
LIN {X 0,Y 375.964,Z 146.655,A -85,B 0,C 180,E1 -12278.271,E2 -12278.271} C_VEL
LIN {X 0,Y 375.926,Z 146.656,A -85,B 0,C 180,E1 -12281.602,E2 -12281.602} C_VEL
LIN {X 0,Y 375.92,Z 146.656,A -85,B 0,C 180,E1 -12285.27,E2 -12285.27} C_VEL
LIN {X 0,Y 375.929,Z 146.658,A -85,B 0,C 180,E1 -12288.4,E2 -12288.4} C_VEL
LIN {X 0,Y 375.969,Z 146.652,A -85,B 0,C 180,E1 -12291.731,E2 -12291.731} C_VEL
LIN {X 0,Y 375.975,Z 146.649,A -85,B 0,C 180,E1 -12295.334,E2 -12295.334} C_VEL
LIN {X 0,Y 375.954,Z 146.658,A -85,B 0,C 180,E1 -12298.439,E2 -12298.439} C_VEL
LIN {X 0,Y 375.99,Z 146.703,A -85,B 0,C 180,E1 -12300.732,E2 -12300.732} C_VEL
LIN {X 0,Y 378.13,Z 157.048,A -85,B 0,C 180,E1 -12303.143,E2 -12303.143} C_VEL
LIN {X 0,Y 379.338,Z 164.313,A -85,B 0,C 180,E1 -12304.78,E2 -12304.78} C_VEL
LIN {X 0,Y 378.068,Z 180.602,A -85,B 0,C 180,E1 -12308.176,E2 -12308.176} C_VEL
LIN {X 0,Y 377.663,Z 185.871,A -85,B 0,C 180,E1 -12309.266,E2 -12309.266} C_VEL
LIN {X 0,Y 382.287,Z 219.322,A -85,B 0,C 180,E1 -12310.159,E2 -12310.159} C_VEL
LIN {X 0,Y 381.303,Z 294.996,A -85,B 0,C 180,E1 -12311.602,E2 -12311.602} C_VEL
LIN {X 0,Y 380.68,Z 308.197,A -85,B 0,C 180,E1 -12312.058,E2 -12312.058} C_VEL
LIN {X 0,Y 379.949,Z 320.919,A -85,B 0,C 180,E1 -12312.717,E2 -12312.717} C_VEL
LIN {X 0,Y 379.052,Z 333.005,A -85,B 0,C 180,E1 -12313.577,E2 -12313.577} C_VEL
LIN {X 0,Y 378.111,Z 344.554,A -85,B 0,C 180,E1 -12314.642,E2 -12314.642} C_VEL
LIN {X 0,Y 377.301,Z 354.314,A -85,B 0,C 180,E1 -12315.767,E2 -12315.767} C_VEL
LIN {X 0,Y 376.467,Z 363.466,A -85,B 0,C 180,E1 -12317.056,E2 -12317.056} C_VEL
LIN {X 0,Y 375.695,Z 372.68,A -85,B 0,C 180,E1 -12318.673,E2 -12318.673} C_VEL
LIN {X 0,Y 375.145,Z 380.1,A -85,B 0,C 180,E1 -12320.294,E2 -12320.294} C_VEL
LIN {X 0,Y 374.824,Z 386.053,A -85,B 0,C 180,E1 -12321.917,E2 -12321.917} C_VEL
LIN {X 0,Y 374.622,Z 390.741,A -85,B 0,C 180,E1 -12323.538,E2 -12323.538} C_VEL
LIN {X 0,Y 374.563,Z 394.309,A -85,B 0,C 180,E1 -12325.158,E2 -12325.158} C_VEL
LIN {X 0,Y 374.526,Z 396.854,A -85,B 0,C 180,E1 -12326.774,E2 -12326.774} C_VEL
LIN {X 0,Y 374.595,Z 398.045,A -85,B 0,C 180,E1 -12327.851,E2 -12327.851} C_VEL
LIN {X 0,Y 374.628,Z 398.787,A -85,B 0,C 180,E1 -12328.926,E2 -12328.926} C_VEL
LIN {X 0,Y 374.613,Z 399.133,A -85,B 0,C 180,E1 -12330.001,E2 -12330.001} C_VEL
LIN {X 0,Y 374.625,Z 399.093,A -85,B 0,C 180,E1 -12331.076,E2 -12331.076} C_VEL
LIN {X 0,Y 374.553,Z 398.659,A -85,B 0,C 180,E1 -12332.152,E2 -12332.152} C_VEL
LIN {X 0,Y 374.549,Z 396.52,A -85,B 0,C 180,E1 -12334.305,E2 -12334.305} C_VEL
LIN {X 0,Y 374.54,Z 393.673,A -85,B 0,C 180,E1 -12336.004,E2 -12336.004} C_VEL
LIN {X 0,Y 374.857,Z 388.69,A -85,B 0,C 180,E1 -12338.084,E2 -12338.084} C_VEL
LIN {X 0,Y 375.322,Z 382.477,A -85,B 0,C 180,E1 -12339.975,E2 -12339.975} C_VEL
LIN {X 0,Y 375.97,Z 375.73,A -85,B 0,C 180,E1 -12341.593,E2 -12341.593} C_VEL
LIN {X 0,Y 377.02,Z 367.383,A -85,B 0,C 180,E1 -12343.201,E2 -12343.201} C_VEL
LIN {X 0,Y 377.895,Z 358.228,A -85,B 0,C 180,E1 -12344.623,E2 -12344.623} C_VEL
LIN {X 0,Y 378.955,Z 348.254,A -85,B 0,C 180,E1 -12345.876,E2 -12345.876} C_VEL
LIN {X 0,Y 380.116,Z 337.814,A -85,B 0,C 180,E1 -12346.931,E2 -12346.931} C_VEL
LIN {X 0,Y 381.235,Z 326.343,A -85,B 0,C 180,E1 -12347.848,E2 -12347.848} C_VEL
LIN {X 0,Y 382.245,Z 314.474,A -85,B 0,C 180,E1 -12348.561,E2 -12348.561} C_VEL
LIN {X 0,Y 382.957,Z 302.604,A -85,B 0,C 180,E1 -12349.081,E2 -12349.081} C_VEL
LIN {X 0,Y 383.443,Z 289.783,A -85,B 0,C 180,E1 -12349.442,E2 -12349.442} C_VEL
LIN {X 0,Y 384.442,Z 219.073,A -85,B 0,C 180,E1 -12350.783,E2 -12350.783} C_VEL
LIN {X 0,Y 380.039,Z 192.502,A -85,B 0,C 180,E1 -12351.591,E2 -12351.591} C_VEL
LIN {X 0,Y 378.644,Z 185.622,A -85,B 0,C 180,E1 -12351.827,E2 -12351.827} C_VEL
LIN {X 0,Y 380.188,Z 169.856,A -85,B 0,C 180,E1 -12355.162,E2 -12355.162} C_VEL
LIN {X 0,Y 380.146,Z 165.863,A -85,B 0,C 180,E1 -12356.046,E2 -12356.046} C_VEL
LIN {X 0,Y 377.616,Z 153.626,A -85,B 0,C 180,E1 -12358.986,E2 -12358.986} C_VEL
LIN {X 0,Y 375.949,Z 146.663,A -85,B 0,C 180,E1 -12360.769,E2 -12360.769} C_VEL
LIN {X 0,Y 375.963,Z 146.655,A -85,B 0,C 180,E1 -12364.112,E2 -12364.112} C_VEL
LIN {X 0,Y 375.955,Z 146.65,A -85,B 0,C 180,E1 -12366.742,E2 -12366.742} C_VEL
LIN {X 0,Y 375.978,Z 146.651,A -85,B 0,C 180,E1 -12369.968,E2 -12369.968} C_VEL
LIN {X 0,Y 375.932,Z 146.657,A -85,B 0,C 180,E1 -12373.766,E2 -12373.766} C_VEL
LIN {X 0,Y 375.936,Z 146.657,A -85,B 0,C 180,E1 -12376.811,E2 -12376.811} C_VEL
LIN {X 0,Y 375.936,Z 146.656,A -85,B 0,C 180,E1 -12380.534,E2 -12380.534} C_VEL
LIN {X 0,Y 375.96,Z 146.656,A -85,B 0,C 180,E1 -12383.497,E2 -12383.497} C_VEL
LIN {X 0,Y 375.959,Z 146.653,A -85,B 0,C 180,E1 -12385.888,E2 -12385.888} C_VEL
LIN {X 0,Y 375.963,Z 146.652,A -85,B 0,C 180,E1 -12389.687,E2 -12389.687} C_VEL
LIN {X 0,Y 375.929,Z 146.655,A -85,B 0,C 180,E1 -12392.136,E2 -12392.136} C_VEL
LIN {X 0,Y 375.969,Z 146.65,A -85,B 0,C 180,E1 -12395.717,E2 -12395.717} C_VEL
LIN {X 0,Y 375.961,Z 146.648,A -85,B 0,C 180,E1 -12399.196,E2 -12399.196} C_VEL
LIN {X 0,Y 376.01,Z 146.649,A -85,B 0,C 180,E1 -12402.599,E2 -12402.599} C_VEL
LIN {X 0,Y 376.092,Z 146.63,A -85,B 0,C 180,E1 -12406.342,E2 -12406.342} C_VEL
LIN {X 0,Y 376.106,Z 146.63,A -85,B 0,C 180,E1 -12410.318,E2 -12410.318} C_VEL
LIN {X 0,Y 376.192,Z 146.622,A -85,B 0,C 180,E1 -12413.564,E2 -12413.564} C_VEL
LIN {X 0,Y 376.331,Z 146.599,A -85,B 0,C 180,E1 -12417.86,E2 -12417.86} C_VEL
LIN {X 0,Y 376.333,Z 146.599,A -85,B 0,C 180,E1 -12422.141,E2 -12422.141} C_VEL
LIN {X 0,Y 376.198,Z 146.621,A -85,B 0,C 180,E1 -12426.436,E2 -12426.436} C_VEL
LIN {X 0,Y 376.114,Z 146.63,A -85,B 0,C 180,E1 -12429.682,E2 -12429.682} C_VEL
LIN {X 0,Y 376.091,Z 146.629,A -85,B 0,C 180,E1 -12433.658,E2 -12433.658} C_VEL
LIN {X 0,Y 376.034,Z 146.645,A -85,B 0,C 180,E1 -12437.4,E2 -12437.4} C_VEL
LIN {X 0,Y 375.981,Z 146.647,A -85,B 0,C 180,E1 -12440.832,E2 -12440.832} C_VEL
LIN {X 0,Y 375.974,Z 146.644,A -85,B 0,C 180,E1 -12444.283,E2 -12444.283} C_VEL
LIN {X 0,Y 375.96,Z 146.649,A -85,B 0,C 180,E1 -12447.862,E2 -12447.862} C_VEL
LIN {X 0,Y 375.959,Z 146.651,A -85,B 0,C 180,E1 -12451.562,E2 -12451.562} C_VEL
LIN {X 0,Y 375.96,Z 146.65,A -85,B 0,C 180,E1 -12455.416,E2 -12455.416} C_VEL
LIN {X 0,Y 375.974,Z 146.652,A -85,B 0,C 180,E1 -12458.27,E2 -12458.27} C_VEL
LIN {X 0,Y 375.937,Z 146.641,A -85,B 0,C 180,E1 -12461.601,E2 -12461.601} C_VEL
LIN {X 0,Y 375.93,Z 146.654,A -85,B 0,C 180,E1 -12465.269,E2 -12465.269} C_VEL
LIN {X 0,Y 375.929,Z 146.661,A -85,B 0,C 180,E1 -12468.401,E2 -12468.401} C_VEL
LIN {X 0,Y 375.974,Z 146.652,A -85,B 0,C 180,E1 -12471.73,E2 -12471.73} C_VEL
LIN {X 0,Y 375.984,Z 146.651,A -85,B 0,C 180,E1 -12475.332,E2 -12475.332} C_VEL
LIN {X 0,Y 375.962,Z 146.651,A -85,B 0,C 180,E1 -12478.438,E2 -12478.438} C_VEL
LIN {X 0,Y 375.998,Z 146.656,A -85,B 0,C 180,E1 -12481,E2 -12481} C_VEL
LIN {X 0,Y 377.769,Z 154.521,A -85,B 0,C 180,E1 -12483.157,E2 -12483.157} C_VEL
LIN {X 0,Y 383.088,Z 168.601,A -85,B 0,C 180,E1 -12483.804,E2 -12483.804} C_VEL
LIN {X 0,Y 385.298,Z 178.844,A -85,B 0,C 180,E1 -12484.15,E2 -12484.15} C_VEL
LIN {X 0,Y 383.83,Z 262.211,A -85,B 0,C 180,E1 -12485.742,E2 -12485.742} C_VEL
LIN {X 0,Y 383.196,Z 275.88,A -85,B 0,C 180,E1 -12486.226,E2 -12486.226} C_VEL
LIN {X 0,Y 382.48,Z 288.614,A -85,B 0,C 180,E1 -12486.91,E2 -12486.91} C_VEL
LIN {X 0,Y 381.59,Z 300.886,A -85,B 0,C 180,E1 -12487.817,E2 -12487.817} C_VEL
LIN {X 0,Y 380.482,Z 312.212,A -85,B 0,C 180,E1 -12488.887,E2 -12488.887} C_VEL
LIN {X 0,Y 379.457,Z 322.369,A -85,B 0,C 180,E1 -12490.102,E2 -12490.102} C_VEL
LIN {X 0,Y 378.415,Z 332.312,A -85,B 0,C 180,E1 -12491.595,E2 -12491.595} C_VEL
LIN {X 0,Y 377.349,Z 341.029,A -85,B 0,C 180,E1 -12493.22,E2 -12493.22} C_VEL
LIN {X 0,Y 376.49,Z 347.949,A -85,B 0,C 180,E1 -12494.85,E2 -12494.85} C_VEL
LIN {X 0,Y 375.843,Z 353.523,A -85,B 0,C 180,E1 -12496.5,E2 -12496.5} C_VEL
LIN {X 0,Y 375.358,Z 357.784,A -85,B 0,C 180,E1 -12498.114,E2 -12498.114} C_VEL
LIN {X 0,Y 375.044,Z 360.063,A -85,B 0,C 180,E1 -12499.199,E2 -12499.199} C_VEL
LIN {X 0,Y 374.877,Z 361.902,A -85,B 0,C 180,E1 -12500.285,E2 -12500.285} C_VEL
LIN {X 0,Y 374.727,Z 364.242,A -85,B 0,C 180,E1 -12502.455,E2 -12502.455} C_VEL
LIN {X 0,Y 374.746,Z 364.894,A -85,B 0,C 180,E1 -12503.705,E2 -12503.705} C_VEL
LIN {X 0,Y 374.62,Z 364.795,A -85,B 0,C 180,E1 -12505.695,E2 -12505.695} C_VEL
LIN {X 0,Y 374.692,Z 363.185,A -85,B 0,C 180,E1 -12507.849,E2 -12507.849} C_VEL
LIN {X 0,Y 374.697,Z 361.797,A -85,B 0,C 180,E1 -12508.924,E2 -12508.924} C_VEL
LIN {X 0,Y 374.898,Z 358.888,A -85,B 0,C 180,E1 -12510.536,E2 -12510.536} C_VEL
LIN {X 0,Y 375.121,Z 354.963,A -85,B 0,C 180,E1 -12512.146,E2 -12512.146} C_VEL
LIN {X 0,Y 375.598,Z 349.9,A -85,B 0,C 180,E1 -12513.754,E2 -12513.754} C_VEL
LIN {X 0,Y 376.127,Z 343.535,A -85,B 0,C 180,E1 -12515.36,E2 -12515.36} C_VEL
LIN {X 0,Y 376.938,Z 335.598,A -85,B 0,C 180,E1 -12516.96,E2 -12516.96} C_VEL
LIN {X 0,Y 377.705,Z 327.511,A -85,B 0,C 180,E1 -12518.29,E2 -12518.29} C_VEL
LIN {X 0,Y 378.606,Z 317.651,A -85,B 0,C 180,E1 -12519.616,E2 -12519.616} C_VEL
LIN {X 0,Y 379.436,Z 306.344,A -85,B 0,C 180,E1 -12520.825,E2 -12520.825} C_VEL
LIN {X 0,Y 380.349,Z 293.871,A -85,B 0,C 180,E1 -12521.861,E2 -12521.861} C_VEL
LIN {X 0,Y 380.831,Z 283.888,A -85,B 0,C 180,E1 -12522.503,E2 -12522.503} C_VEL
LIN {X 0,Y 380.539,Z 278.388,A -85,B 0,C 180,E1 -12522.825,E2 -12522.825} C_VEL
LIN {X 0,Y 378.096,Z 269.378,A -85,B 0,C 180,E1 -12523.334,E2 -12523.334} C_VEL
LIN {X 0,Y 375.508,Z 260.181,A -85,B 0,C 180,E1 -12523.742,E2 -12523.742} C_VEL
LIN {X 0,Y 374.974,Z 254.389,A -85,B 0,C 180,E1 -12523.897,E2 -12523.897} C_VEL
LIN {X 0,Y 376.098,Z 177.371,A -85,B 0,C 180,E1 -12525.36,E2 -12525.36} C_VEL
LIN {X 0,Y 372.755,Z 161.261,A -85,B 0,C 180,E1 -12525.856,E2 -12525.856} C_VEL
LIN {X 0,Y 370.404,Z 154.492,A -85,B 0,C 180,E1 -12526.136,E2 -12526.136} C_VEL
LIN {X 0,Y 369.008,Z 147.52,A -85,B 0,C 180,E1 -12527.998,E2 -12527.998} C_VEL
LIN {X 0,Y 368.909,Z 147.529,A -85,B 0,C 180,E1 -12531.219,E2 -12531.219} C_VEL
LIN {X 0,Y 368.954,Z 147.525,A -85,B 0,C 180,E1 -12534.774,E2 -12534.774} C_VEL
LIN {X 0,Y 368.967,Z 147.521,A -85,B 0,C 180,E1 -12537.202,E2 -12537.202} C_VEL
LIN {X 0,Y 368.917,Z 147.529,A -85,B 0,C 180,E1 -12539.689,E2 -12539.689} C_VEL
LIN {X 0,Y 368.894,Z 147.531,A -85,B 0,C 180,E1 -12543.042,E2 -12543.042} C_VEL
LIN {X 0,Y 368.914,Z 147.533,A -85,B 0,C 180,E1 -12546.195,E2 -12546.195} C_VEL
LIN {X 0,Y 368.899,Z 147.53,A -85,B 0,C 180,E1 -12548.952,E2 -12548.952} C_VEL
LIN {X 0,Y 368.877,Z 147.538,A -85,B 0,C 180,E1 -12552.008,E2 -12552.008} C_VEL
LIN {X 0,Y 368.874,Z 147.534,A -85,B 0,C 180,E1 -12555.174,E2 -12555.174} C_VEL
LIN {X 0,Y 368.876,Z 147.536,A -85,B 0,C 180,E1 -12558.176,E2 -12558.176} C_VEL
LIN {X 0,Y 368.899,Z 147.532,A -85,B 0,C 180,E1 -12561.359,E2 -12561.359} C_VEL
LIN {X 0,Y 368.928,Z 147.528,A -85,B 0,C 180,E1 -12565.145,E2 -12565.145} C_VEL
LIN {X 0,Y 368.921,Z 147.529,A -85,B 0,C 180,E1 -12569.045,E2 -12569.045} C_VEL
LIN {X 0,Y 368.967,Z 147.528,A -85,B 0,C 180,E1 -12571.563,E2 -12571.563} C_VEL
LIN {X 0,Y 368.935,Z 147.529,A -85,B 0,C 180,E1 -12575.223,E2 -12575.223} C_VEL
LIN {X 0,Y 368.91,Z 147.531,A -85,B 0,C 180,E1 -12578.98,E2 -12578.98} C_VEL
LIN {X 0,Y 368.981,Z 147.52,A -85,B 0,C 180,E1 -12582.256,E2 -12582.256} C_VEL
LIN {X 0,Y 369.027,Z 147.514,A -85,B 0,C 180,E1 -12586.227,E2 -12586.227} C_VEL
LIN {X 0,Y 369.051,Z 147.511,A -85,B 0,C 180,E1 -12590.131,E2 -12590.131} C_VEL
LIN {X 0,Y 369.143,Z 147.504,A -85,B 0,C 180,E1 -12593.441,E2 -12593.441} C_VEL
LIN {X 0,Y 369.288,Z 147.482,A -85,B 0,C 180,E1 -12597.819,E2 -12597.819} C_VEL
LIN {X 0,Y 369.289,Z 147.482,A -85,B 0,C 180,E1 -12602.181,E2 -12602.181} C_VEL
LIN {X 0,Y 369.148,Z 147.502,A -85,B 0,C 180,E1 -12606.559,E2 -12606.559} C_VEL
LIN {X 0,Y 369.051,Z 147.511,A -85,B 0,C 180,E1 -12609.869,E2 -12609.869} C_VEL
LIN {X 0,Y 369.026,Z 147.514,A -85,B 0,C 180,E1 -12613.772,E2 -12613.772} C_VEL
LIN {X 0,Y 368.98,Z 147.52,A -85,B 0,C 180,E1 -12617.743,E2 -12617.743} C_VEL
LIN {X 0,Y 368.899,Z 147.531,A -85,B 0,C 180,E1 -12621.221,E2 -12621.221} C_VEL
LIN {X 0,Y 368.934,Z 147.53,A -85,B 0,C 180,E1 -12624.777,E2 -12624.777} C_VEL
LIN {X 0,Y 368.97,Z 147.527,A -85,B 0,C 180,E1 -12628.437,E2 -12628.437} C_VEL
LIN {X 0,Y 368.889,Z 147.536,A -85,B 0,C 180,E1 -12632.239,E2 -12632.239} C_VEL
LIN {X 0,Y 368.92,Z 147.528,A -85,B 0,C 180,E1 -12635.002,E2 -12635.002} C_VEL
LIN {X 0,Y 368.899,Z 147.533,A -85,B 0,C 180,E1 -12638.641,E2 -12638.641} C_VEL
LIN {X 0,Y 368.874,Z 147.537,A -85,B 0,C 180,E1 -12642.011,E2 -12642.011} C_VEL
LIN {X 0,Y 368.873,Z 147.533,A -85,B 0,C 180,E1 -12645.177,E2 -12645.177} C_VEL
LIN {X 0,Y 368.877,Z 147.539,A -85,B 0,C 180,E1 -12648.179,E2 -12648.179} C_VEL
LIN {X 0,Y 368.904,Z 147.53,A -85,B 0,C 180,E1 -12651.361,E2 -12651.361} C_VEL
LIN {X 0,Y 368.932,Z 147.526,A -85,B 0,C 180,E1 -12655.148,E2 -12655.148} C_VEL
LIN {X 0,Y 368.926,Z 147.533,A -85,B 0,C 180,E1 -12659.048,E2 -12659.048} C_VEL
LIN {X 0,Y 368.962,Z 147.721,A -85,B 0,C 180,E1 -12660.476,E2 -12660.476} C_VEL
LIN {X 0,Y 371.158,Z 158.201,A -85,B 0,C 180,E1 -12662.972,E2 -12662.972} C_VEL
LIN {X 0,Y 372.379,Z 165.759,A -85,B 0,C 180,E1 -12664.706,E2 -12664.706} C_VEL
LIN {X 0,Y 371.007,Z 182.021,A -85,B 0,C 180,E1 -12668.158,E2 -12668.158} C_VEL
LIN {X 0,Y 370.761,Z 185.614,A -85,B 0,C 180,E1 -12668.917,E2 -12668.917} C_VEL
LIN {X 0,Y 375.516,Z 220.01,A -85,B 0,C 180,E1 -12669.844,E2 -12669.844} C_VEL
LIN {X 0,Y 374.497,Z 294.601,A -85,B 0,C 180,E1 -12671.291,E2 -12671.291} C_VEL
LIN {X 0,Y 373.87,Z 307.83,A -85,B 0,C 180,E1 -12671.755,E2 -12671.755} C_VEL
LIN {X 0,Y 373.172,Z 319.998,A -85,B 0,C 180,E1 -12672.393,E2 -12672.393} C_VEL
LIN {X 0,Y 372.204,Z 332.26,A -85,B 0,C 180,E1 -12673.266,E2 -12673.266} C_VEL
LIN {X 0,Y 371.21,Z 343.883,A -85,B 0,C 180,E1 -12674.349,E2 -12674.349} C_VEL
LIN {X 0,Y 370.284,Z 354.73,A -85,B 0,C 180,E1 -12675.625,E2 -12675.625} C_VEL
LIN {X 0,Y 369.376,Z 364.584,A -85,B 0,C 180,E1 -12677.083,E2 -12677.083} C_VEL
LIN {X 0,Y 368.565,Z 373.544,A -85,B 0,C 180,E1 -12678.73,E2 -12678.73} C_VEL
LIN {X 0,Y 368.048,Z 380.745,A -85,B 0,C 180,E1 -12680.383,E2 -12680.383} C_VEL
LIN {X 0,Y 367.663,Z 387.297,A -85,B 0,C 180,E1 -12682.311,E2 -12682.311} C_VEL
LIN {X 0,Y 367.514,Z 391.558,A -85,B 0,C 180,E1 -12683.935,E2 -12683.935} C_VEL
LIN {X 0,Y 367.5,Z 394.873,A -85,B 0,C 180,E1 -12685.614,E2 -12685.614} C_VEL
LIN {X 0,Y 367.495,Z 397.689,A -85,B 0,C 180,E1 -12687.809,E2 -12687.809} C_VEL
LIN {X 0,Y 367.543,Z 398.448,A -85,B 0,C 180,E1 -12688.905,E2 -12688.905} C_VEL
LIN {X 0,Y 367.546,Z 398.805,A -85,B 0,C 180,E1 -12690.001,E2 -12690.001} C_VEL
LIN {X 0,Y 367.539,Z 398.774,A -85,B 0,C 180,E1 -12691.097,E2 -12691.097} C_VEL
LIN {X 0,Y 367.453,Z 398.353,A -85,B 0,C 180,E1 -12692.193,E2 -12692.193} C_VEL
LIN {X 0,Y 367.407,Z 397.501,A -85,B 0,C 180,E1 -12693.291,E2 -12693.291} C_VEL
LIN {X 0,Y 367.453,Z 396.241,A -85,B 0,C 180,E1 -12694.389,E2 -12694.389} C_VEL
LIN {X 0,Y 367.461,Z 393.68,A -85,B 0,C 180,E1 -12695.986,E2 -12695.986} C_VEL
LIN {X 0,Y 367.675,Z 389.904,A -85,B 0,C 180,E1 -12697.69,E2 -12697.69} C_VEL
LIN {X 0,Y 368.041,Z 385.128,A -85,B 0,C 180,E1 -12699.342,E2 -12699.342} C_VEL
LIN {X 0,Y 368.744,Z 377.985,A -85,B 0,C 180,E1 -12701.266,E2 -12701.266} C_VEL
LIN {X 0,Y 369.724,Z 370.238,A -85,B 0,C 180,E1 -12702.907,E2 -12702.907} C_VEL
LIN {X 0,Y 370.698,Z 360.901,A -85,B 0,C 180,E1 -12704.494,E2 -12704.494} C_VEL
LIN {X 0,Y 371.872,Z 350.561,A -85,B 0,C 180,E1 -12705.905,E2 -12705.905} C_VEL
LIN {X 0,Y 373.149,Z 339.293,A -85,B 0,C 180,E1 -12707.115,E2 -12707.115} C_VEL
LIN {X 0,Y 374.332,Z 328.271,A -85,B 0,C 180,E1 -12708.047,E2 -12708.047} C_VEL
LIN {X 0,Y 375.445,Z 316.062,A -85,B 0,C 180,E1 -12708.839,E2 -12708.839} C_VEL
LIN {X 0,Y 376.224,Z 304.169,A -85,B 0,C 180,E1 -12709.401,E2 -12709.401} C_VEL
LIN {X 0,Y 376.808,Z 290.988,A -85,B 0,C 180,E1 -12709.8,E2 -12709.8} C_VEL
LIN {X 0,Y 377.905,Z 219.971,A -85,B 0,C 180,E1 -12711.173,E2 -12711.173} C_VEL
LIN {X 0,Y 373.527,Z 193.798,A -85,B 0,C 180,E1 -12711.993,E2 -12711.993} C_VEL
LIN {X 0,Y 371.855,Z 185.297,A -85,B 0,C 180,E1 -12712.284,E2 -12712.284} C_VEL
LIN {X 0,Y 373.465,Z 169.713,A -85,B 0,C 180,E1 -12715.648,E2 -12715.648} C_VEL
LIN {X 0,Y 372.402,Z 163.011,A -85,B 0,C 180,E1 -12717.242,E2 -12717.242} C_VEL
LIN {X 0,Y 369.71,Z 150.997,A -85,B 0,C 180,E1 -12720.249,E2 -12720.249} C_VEL
LIN {X 0,Y 368.918,Z 147.537,A -85,B 0,C 180,E1 -12721.186,E2 -12721.186} C_VEL
LIN {X 0,Y 368.931,Z 147.527,A -85,B 0,C 180,E1 -12725.002,E2 -12725.002} C_VEL
LIN {X 0,Y 368.905,Z 147.529,A -85,B 0,C 180,E1 -12728.639,E2 -12728.639} C_VEL
LIN {X 0,Y 368.881,Z 147.534,A -85,B 0,C 180,E1 -12732.009,E2 -12732.009} C_VEL
LIN {X 0,Y 368.881,Z 147.537,A -85,B 0,C 180,E1 -12735.176,E2 -12735.176} C_VEL
LIN {X 0,Y 368.872,Z 147.536,A -85,B 0,C 180,E1 -12738.176,E2 -12738.176} C_VEL
LIN {X 0,Y 368.878,Z 147.538,A -85,B 0,C 180,E1 -12741.366,E2 -12741.366} C_VEL
LIN {X 0,Y 368.932,Z 147.531,A -85,B 0,C 180,E1 -12745.146,E2 -12745.146} C_VEL
LIN {X 0,Y 368.914,Z 147.533,A -85,B 0,C 180,E1 -12749.045,E2 -12749.045} C_VEL
LIN {X 0,Y 368.913,Z 147.529,A -85,B 0,C 180,E1 -12751.558,E2 -12751.558} C_VEL
LIN {X 0,Y 368.924,Z 147.53,A -85,B 0,C 180,E1 -12755.222,E2 -12755.222} C_VEL
LIN {X 0,Y 368.921,Z 147.526,A -85,B 0,C 180,E1 -12758.981,E2 -12758.981} C_VEL
LIN {X 0,Y 368.954,Z 147.524,A -85,B 0,C 180,E1 -12762.255,E2 -12762.255} C_VEL
LIN {X 0,Y 369.039,Z 147.507,A -85,B 0,C 180,E1 -12766.228,E2 -12766.228} C_VEL
LIN {X 0,Y 369.057,Z 147.51,A -85,B 0,C 180,E1 -12770.132,E2 -12770.132} C_VEL
LIN {X 0,Y 369.154,Z 147.498,A -85,B 0,C 180,E1 -12773.441,E2 -12773.441} C_VEL
LIN {X 0,Y 369.294,Z 147.475,A -85,B 0,C 180,E1 -12777.819,E2 -12777.819} C_VEL
LIN {X 0,Y 369.202,Z 147.493,A -85,B 0,C 180,E1 -12781.091,E2 -12781.091} C_VEL
LIN {X 0,Y 369.296,Z 147.475,A -85,B 0,C 180,E1 -12782.181,E2 -12782.181} C_VEL
LIN {X 0,Y 369.159,Z 147.498,A -85,B 0,C 180,E1 -12786.559,E2 -12786.559} C_VEL
LIN {X 0,Y 369.064,Z 147.51,A -85,B 0,C 180,E1 -12789.869,E2 -12789.869} C_VEL
LIN {X 0,Y 369.039,Z 147.507,A -85,B 0,C 180,E1 -12793.772,E2 -12793.772} C_VEL
LIN {X 0,Y 368.993,Z 147.519,A -85,B 0,C 180,E1 -12797.743,E2 -12797.743} C_VEL
LIN {X 0,Y 368.912,Z 147.532,A -85,B 0,C 180,E1 -12801.221,E2 -12801.221} C_VEL
LIN {X 0,Y 368.93,Z 147.523,A -85,B 0,C 180,E1 -12804.778,E2 -12804.778} C_VEL
LIN {X 0,Y 368.933,Z 147.526,A -85,B 0,C 180,E1 -12808.44,E2 -12808.44} C_VEL
LIN {X 0,Y 368.913,Z 147.533,A -85,B 0,C 180,E1 -12810.987,E2 -12810.987} C_VEL
LIN {X 0,Y 368.939,Z 147.529,A -85,B 0,C 180,E1 -12814.854,E2 -12814.854} C_VEL
LIN {X 0,Y 368.909,Z 147.531,A -85,B 0,C 180,E1 -12818.64,E2 -12818.64} C_VEL
LIN {X 0,Y 368.884,Z 147.521,A -85,B 0,C 180,E1 -12822.009,E2 -12822.009} C_VEL
LIN {X 0,Y 368.883,Z 147.532,A -85,B 0,C 180,E1 -12825.176,E2 -12825.176} C_VEL
LIN {X 0,Y 368.879,Z 147.537,A -85,B 0,C 180,E1 -12828.177,E2 -12828.177} C_VEL
LIN {X 0,Y 368.908,Z 147.531,A -85,B 0,C 180,E1 -12831.36,E2 -12831.36} C_VEL
LIN {X 0,Y 368.94,Z 147.528,A -85,B 0,C 180,E1 -12835.146,E2 -12835.146} C_VEL
LIN {X 0,Y 368.933,Z 147.528,A -85,B 0,C 180,E1 -12839.046,E2 -12839.046} C_VEL
LIN {X 0,Y 368.97,Z 147.72,A -85,B 0,C 180,E1 -12840.667,E2 -12840.667} C_VEL
LIN {X 0,Y 370.607,Z 154.959,A -85,B 0,C 180,E1 -12842.678,E2 -12842.678} C_VEL
LIN {X 0,Y 376.704,Z 170.502,A -85,B 0,C 180,E1 -12843.42,E2 -12843.42} C_VEL
LIN {X 0,Y 378.764,Z 179.749,A -85,B 0,C 180,E1 -12843.745,E2 -12843.745} C_VEL
LIN {X 0,Y 377.253,Z 261.691,A -85,B 0,C 180,E1 -12845.328,E2 -12845.328} C_VEL
LIN {X 0,Y 376.65,Z 274.949,A -85,B 0,C 180,E1 -12845.79,E2 -12845.79} C_VEL
LIN {X 0,Y 375.829,Z 287.999,A -85,B 0,C 180,E1 -12846.477,E2 -12846.477} C_VEL
LIN {X 0,Y 375.097,Z 298.921,A -85,B 0,C 180,E1 -12847.266,E2 -12847.266} C_VEL
LIN {X 0,Y 373.982,Z 310.679,A -85,B 0,C 180,E1 -12848.358,E2 -12848.358} C_VEL
LIN {X 0,Y 372.878,Z 320.129,A -85,B 0,C 180,E1 -12849.448,E2 -12849.448} C_VEL
LIN {X 0,Y 371.811,Z 330.409,A -85,B 0,C 180,E1 -12850.928,E2 -12850.928} C_VEL
LIN {X 0,Y 370.87,Z 338.358,A -85,B 0,C 180,E1 -12852.349,E2 -12852.349} C_VEL
LIN {X 0,Y 369.852,Z 345.88,A -85,B 0,C 180,E1 -12854.005,E2 -12854.005} C_VEL
LIN {X 0,Y 369.084,Z 351.901,A -85,B 0,C 180,E1 -12855.667,E2 -12855.667} C_VEL
LIN {X 0,Y 368.484,Z 356.649,A -85,B 0,C 180,E1 -12857.329,E2 -12857.329} C_VEL
LIN {X 0,Y 368.019,Z 360.272,A -85,B 0,C 180,E1 -12858.99,E2 -12858.99} C_VEL
LIN {X 0,Y 367.841,Z 362.136,A -85,B 0,C 180,E1 -12860.098,E2 -12860.098} C_VEL
LIN {X 0,Y 367.702,Z 363.536,A -85,B 0,C 180,E1 -12861.204,E2 -12861.204} C_VEL
LIN {X 0,Y 367.638,Z 365.125,A -85,B 0,C 180,E1 -12863.413,E2 -12863.413} C_VEL
LIN {X 0,Y 367.584,Z 365.347,A -85,B 0,C 180,E1 -12864.513,E2 -12864.513} C_VEL
LIN {X 0,Y 367.548,Z 365.144,A -85,B 0,C 180,E1 -12865.612,E2 -12865.612} C_VEL
LIN {X 0,Y 367.594,Z 363.57,A -85,B 0,C 180,E1 -12867.808,E2 -12867.808} C_VEL
LIN {X 0,Y 367.628,Z 362.206,A -85,B 0,C 180,E1 -12868.904,E2 -12868.904} C_VEL
LIN {X 0,Y 367.808,Z 359.329,A -85,B 0,C 180,E1 -12870.546,E2 -12870.546} C_VEL
LIN {X 0,Y 368.047,Z 355.44,A -85,B 0,C 180,E1 -12872.188,E2 -12872.188} C_VEL
LIN {X 0,Y 368.557,Z 350.423,A -85,B 0,C 180,E1 -12873.826,E2 -12873.826} C_VEL
LIN {X 0,Y 369.098,Z 344.122,A -85,B 0,C 180,E1 -12875.462,E2 -12875.462} C_VEL
LIN {X 0,Y 369.934,Z 336.24,A -85,B 0,C 180,E1 -12877.092,E2 -12877.092} C_VEL
LIN {X 0,Y 370.844,Z 326.456,A -85,B 0,C 180,E1 -12878.719,E2 -12878.719} C_VEL
LIN {X 0,Y 371.827,Z 316.278,A -85,B 0,C 180,E1 -12880.057,E2 -12880.057} C_VEL
LIN {X 0,Y 372.608,Z 306.043,A -85,B 0,C 180,E1 -12881.146,E2 -12881.146} C_VEL
LIN {X 0,Y 373.475,Z 294.947,A -85,B 0,C 180,E1 -12882.083,E2 -12882.083} C_VEL
LIN {X 0,Y 374.078,Z 282.555,A -85,B 0,C 180,E1 -12882.89,E2 -12882.89} C_VEL
LIN {X 0,Y 374.663,Z 270.167,A -85,B 0,C 180,E1 -12883.456,E2 -12883.456} C_VEL
LIN {X 0,Y 374.919,Z 257.754,A -85,B 0,C 180,E1 -12883.827,E2 -12883.827} C_VEL
LIN {X 0,Y 374.974,Z 254.389,A -85,B 0,C 180,E1 -12883.897,E2 -12883.897} C_VEL
LIN {X 0,Y 374.462,Z 248.572,A -85,B 0,C 180,E1 -12884.036,E2 -12884.036} C_VEL
LIN {X 0,Y 369.307,Z 229.836,A -85,B 0,C 180,E1 -12884.662,E2 -12884.662} C_VEL
LIN {X 0,Y 368.76,Z 224.019,A -85,B 0,C 180,E1 -12884.807,E2 -12884.807} C_VEL
LIN {X 0,Y 369.42,Z 178.424,A -85,B 0,C 180,E1 -12885.69,E2 -12885.69} C_VEL
LIN {X 0,Y 366.119,Z 163,A -85,B 0,C 180,E1 -12886.183,E2 -12886.183} C_VEL
LIN {X 0,Y 363.25,Z 154.76,A -85,B 0,C 180,E1 -12886.542,E2 -12886.542} C_VEL
LIN {X 0,Y 361.961,Z 148.4,A -85,B 0,C 180,E1 -12888.317,E2 -12888.317} C_VEL
LIN {X 0,Y 361.861,Z 148.407,A -85,B 0,C 180,E1 -12891.653,E2 -12891.653} C_VEL
LIN {X 0,Y 361.926,Z 148.398,A -85,B 0,C 180,E1 -12895.289,E2 -12895.289} C_VEL
LIN {X 0,Y 361.917,Z 148.402,A -85,B 0,C 180,E1 -12897.777,E2 -12897.777} C_VEL
LIN {X 0,Y 361.844,Z 148.409,A -85,B 0,C 180,E1 -12901.284,E2 -12901.284} C_VEL
LIN {X 0,Y 361.851,Z 148.412,A -85,B 0,C 180,E1 -12904.279,E2 -12904.279} C_VEL
LIN {X 0,Y 361.86,Z 148.407,A -85,B 0,C 180,E1 -12907.222,E2 -12907.222} C_VEL
LIN {X 0,Y 361.831,Z 148.411,A -85,B 0,C 180,E1 -12910.754,E2 -12910.754} C_VEL
LIN {X 0,Y 361.812,Z 148.415,A -85,B 0,C 180,E1 -12914.367,E2 -12914.367} C_VEL
LIN {X 0,Y 361.83,Z 148.414,A -85,B 0,C 180,E1 -12917.567,E2 -12917.567} C_VEL
LIN {X 0,Y 361.861,Z 148.407,A -85,B 0,C 180,E1 -12920.973,E2 -12920.973} C_VEL
